LIN {X 0,Y 421.823,Z 772.372,A -85,B 0,C 180,E1 -10186.267,E2 -10186.267} C_VEL
LIN {X 0,Y 422.37,Z 759.301,A -85,B 0,C 180,E1 -10186.742,E2 -10186.742} C_VEL
LIN {X 0,Y 422.695,Z 742.091,A -85,B 0,C 180,E1 -10187.102,E2 -10187.102} C_VEL
LIN {X 0,Y 423.433,Z 672.26,A -85,B 0,C 180,E1 -10188.345,E2 -10188.345} C_VEL
LIN {X 0,Y 419.664,Z 646.445,A -85,B 0,C 180,E1 -10189.009,E2 -10189.009} C_VEL
LIN {X 0,Y 420.83,Z 628.889,A -85,B 0,C 180,E1 -10192.329,E2 -10192.329} C_VEL
LIN {X 0,Y 421.665,Z 615.532,A -85,B 0,C 180,E1 -10194.887,E2 -10194.887} C_VEL
LIN {X 0,Y 419.461,Z 603.65,A -85,B 0,C 180,E1 -10197.375,E2 -10197.375} C_VEL
LIN {X 0,Y 418.306,Z 598.381,A -85,B 0,C 180,E1 -10198.54,E2 -10198.54} C_VEL
LIN {X 0,Y 418.211,Z 598.39,A -85,B 0,C 180,E1 -10201.395,E2 -10201.395} C_VEL
LIN {X 0,Y 418.266,Z 598.386,A -85,B 0,C 180,E1 -10204.579,E2 -10204.579} C_VEL
LIN {X 0,Y 418.236,Z 598.384,A -85,B 0,C 180,E1 -10207.834,E2 -10207.834} C_VEL
LIN {X 0,Y 418.263,Z 598.383,A -85,B 0,C 180,E1 -10210.942,E2 -10210.942} C_VEL
LIN {X 0,Y 418.207,Z 598.387,A -85,B 0,C 180,E1 -10213.728,E2 -10213.728} C_VEL
LIN {X 0,Y 418.212,Z 598.391,A -85,B 0,C 180,E1 -10216.449,E2 -10216.449} C_VEL
LIN {X 0,Y 418.261,Z 598.383,A -85,B 0,C 180,E1 -10219.123,E2 -10219.123} C_VEL
LIN {X 0,Y 418.231,Z 598.385,A -85,B 0,C 180,E1 -10222.164,E2 -10222.164} C_VEL
LIN {X 0,Y 418.261,Z 598.381,A -85,B 0,C 180,E1 -10225.419,E2 -10225.419} C_VEL
LIN {X 0,Y 418.218,Z 598.389,A -85,B 0,C 180,E1 -10228.604,E2 -10228.604} C_VEL
LIN {X 0,Y 418.289,Z 598.376,A -85,B 0,C 180,E1 -10231.936,E2 -10231.936} C_VEL
LIN {X 0,Y 418.283,Z 598.383,A -85,B 0,C 180,E1 -10235.162,E2 -10235.162} C_VEL
LIN {X 0,Y 418.226,Z 598.385,A -85,B 0,C 180,E1 -10238.303,E2 -10238.303} C_VEL
LIN {X 0,Y 418.276,Z 598.382,A -85,B 0,C 180,E1 -10241.382,E2 -10241.382} C_VEL
LIN {X 0,Y 418.293,Z 598.376,A -85,B 0,C 180,E1 -10244.405,E2 -10244.405} C_VEL
LIN {X 0,Y 418.347,Z 598.375,A -85,B 0,C 180,E1 -10247.385,E2 -10247.385} C_VEL
LIN {X 0,Y 418.334,Z 598.371,A -85,B 0,C 180,E1 -10250.328,E2 -10250.328} C_VEL
LIN {X 0,Y 418.485,Z 598.359,A -85,B 0,C 180,E1 -10253.248,E2 -10253.248} C_VEL
LIN {X 0,Y 418.336,Z 598.376,A -85,B 0,C 180,E1 -10255.181,E2 -10255.181} C_VEL
LIN {X 0,Y 418.535,Z 598.347,A -85,B 0,C 180,E1 -10258.075,E2 -10258.075} C_VEL
LIN {X 0,Y 418.664,Z 598.331,A -85,B 0,C 180,E1 -10260,E2 -10260} C_VEL
LIN {X 0,Y 418.503,Z 598.351,A -85,B 0,C 180,E1 -10262.887,E2 -10262.887} C_VEL
LIN {X 0,Y 418.483,Z 598.352,A -85,B 0,C 180,E1 -10266.64,E2 -10266.64} C_VEL
LIN {X 0,Y 418.348,Z 598.377,A -85,B 0,C 180,E1 -10269.671,E2 -10269.671} C_VEL
LIN {X 0,Y 418.336,Z 598.371,A -85,B 0,C 180,E1 -10273,E2 -10273} C_VEL
LIN {X 0,Y 418.303,Z 598.375,A -85,B 0,C 180,E1 -10276.735,E2 -10276.735} C_VEL
LIN {X 0,Y 418.261,Z 598.388,A -85,B 0,C 180,E1 -10279.79,E2 -10279.79} C_VEL
LIN {X 0,Y 418.228,Z 598.384,A -85,B 0,C 180,E1 -10282.736,E2 -10282.736} C_VEL
LIN {X 0,Y 418.262,Z 598.388,A -85,B 0,C 180,E1 -10285.904,E2 -10285.904} C_VEL
LIN {X 0,Y 418.265,Z 598.38,A -85,B 0,C 180,E1 -10289.161,E2 -10289.161} C_VEL
LIN {X 0,Y 418.251,Z 598.381,A -85,B 0,C 180,E1 -10292.845,E2 -10292.845} C_VEL
LIN {X 0,Y 418.24,Z 598.389,A -85,B 0,C 180,E1 -10296.239,E2 -10296.239} C_VEL
LIN {X 0,Y 418.26,Z 598.382,A -85,B 0,C 180,E1 -10299.68,E2 -10299.68} C_VEL
LIN {X 0,Y 418.278,Z 598.384,A -85,B 0,C 180,E1 -10302.33,E2 -10302.33} C_VEL
LIN {X 0,Y 418.247,Z 598.382,A -85,B 0,C 180,E1 -10305.112,E2 -10305.112} C_VEL
LIN {X 0,Y 418.249,Z 598.383,A -85,B 0,C 180,E1 -10307.769,E2 -10307.769} C_VEL
LIN {X 0,Y 418.253,Z 598.386,A -85,B 0,C 180,E1 -10310.619,E2 -10310.619} C_VEL
LIN {X 0,Y 418.239,Z 598.385,A -85,B 0,C 180,E1 -10313.977,E2 -10313.977} C_VEL
LIN {X 0,Y 418.251,Z 598.382,A -85,B 0,C 180,E1 -10317.156,E2 -10317.156} C_VEL
LIN {X 0,Y 418.263,Z 598.383,A -85,B 0,C 180,E1 -10320.896,E2 -10320.896} C_VEL
LIN {X 0,Y 418.266,Z 598.381,A -85,B 0,C 180,E1 -10324.096,E2 -10324.096} C_VEL
LIN {X 0,Y 418.234,Z 598.385,A -85,B 0,C 180,E1 -10327.264,E2 -10327.264} C_VEL
LIN {X 0,Y 418.279,Z 598.381,A -85,B 0,C 180,E1 -10330.365,E2 -10330.365} C_VEL
LIN {X 0,Y 418.313,Z 598.375,A -85,B 0,C 180,E1 -10333.405,E2 -10333.405} C_VEL
LIN {X 0,Y 418.343,Z 598.376,A -85,B 0,C 180,E1 -10336.999,E2 -10336.999} C_VEL
LIN {X 0,Y 418.338,Z 598.372,A -85,B 0,C 180,E1 -10340.329,E2 -10340.329} C_VEL
LIN {X 0,Y 418.484,Z 598.356,A -85,B 0,C 180,E1 -10343.249,E2 -10343.249} C_VEL
LIN {X 0,Y 418.337,Z 598.376,A -85,B 0,C 180,E1 -10345.182,E2 -10345.182} C_VEL
LIN {X 0,Y 418.542,Z 598.345,A -85,B 0,C 180,E1 -10348.076,E2 -10348.076} C_VEL
LIN {X 0,Y 418.67,Z 598.329,A -85,B 0,C 180,E1 -10350,E2 -10350} C_VEL
LIN {X 0,Y 418.508,Z 598.354,A -85,B 0,C 180,E1 -10352.888,E2 -10352.888} C_VEL
LIN {X 0,Y 418.484,Z 598.355,A -85,B 0,C 180,E1 -10356.751,E2 -10356.751} C_VEL
LIN {X 0,Y 418.338,Z 598.373,A -85,B 0,C 180,E1 -10359.671,E2 -10359.671} C_VEL
LIN {X 0,Y 418.319,Z 598.376,A -85,B 0,C 180,E1 -10363.342,E2 -10363.342} C_VEL
LIN {X 0,Y 417.626,Z 598.464,A -85,B 0,C 180,E1 -10364.146,E2 -10364.146} C_VEL
LIN {X 0,Y 414.748,Z 598.824,A -85,B 0,C 180,E1 -10365.451,E2 -10365.451} C_VEL
LIN {X 0,Y 412.334,Z 599.121,A -85,B 0,C 180,E1 -10366.505,E2 -10366.505} C_VEL
LIN {X 0,Y 411.312,Z 599.253,A -85,B 0,C 180,E1 -10367.32,E2 -10367.32} C_VEL
LIN {X 0,Y 411.236,Z 599.257,A -85,B 0,C 180,E1 -10367.596,E2 -10367.596} C_VEL
LIN {X 0,Y 411.195,Z 599.266,A -85,B 0,C 180,E1 -10371.034,E2 -10371.034} C_VEL
LIN {X 0,Y 411.276,Z 599.382,A -85,B 0,C 180,E1 -10373.276,E2 -10373.276} C_VEL
LIN {X 0,Y 412.939,Z 608.733,A -85,B 0,C 180,E1 -10375.742,E2 -10375.742} C_VEL
LIN {X 0,Y 412.98,Z 609.152,A -85,B 0,C 180,E1 -10375.806,E2 -10375.806} C_VEL
LIN {X 0,Y 417.05,Z 628.232,A -85,B 0,C 180,E1 -10376.355,E2 -10376.355} C_VEL
LIN {X 0,Y 415.798,Z 716.325,A -85,B 0,C 180,E1 -10377.971,E2 -10377.971} C_VEL
LIN {X 0,Y 415.423,Z 730.048,A -85,B 0,C 180,E1 -10378.435,E2 -10378.435} C_VEL
LIN {X 0,Y 414.909,Z 742.373,A -85,B 0,C 180,E1 -10379.048,E2 -10379.048} C_VEL
LIN {X 0,Y 414.304,Z 753.409,A -85,B 0,C 180,E1 -10379.782,E2 -10379.782} C_VEL
LIN {X 0,Y 413.557,Z 765.254,A -85,B 0,C 180,E1 -10380.793,E2 -10380.793} C_VEL
LIN {X 0,Y 412.878,Z 775.146,A -85,B 0,C 180,E1 -10381.848,E2 -10381.848} C_VEL
LIN {X 0,Y 412.252,Z 784.368,A -85,B 0,C 180,E1 -10383.06,E2 -10383.06} C_VEL
LIN {X 0,Y 411.647,Z 792.069,A -85,B 0,C 180,E1 -10384.291,E2 -10384.291} C_VEL
LIN {X 0,Y 411.086,Z 799.616,A -85,B 0,C 180,E1 -10385.772,E2 -10385.772} C_VEL
LIN {X 0,Y 410.669,Z 806.242,A -85,B 0,C 180,E1 -10387.41,E2 -10387.41} C_VEL
LIN {X 0,Y 410.42,Z 810.287,A -85,B 0,C 180,E1 -10388.682,E2 -10388.682} C_VEL
LIN {X 0,Y 410.182,Z 813.761,A -85,B 0,C 180,E1 -10390.061,E2 -10390.061} C_VEL
LIN {X 0,Y 410.086,Z 815.725,A -85,B 0,C 180,E1 -10391.057,E2 -10391.057} C_VEL
LIN {X 0,Y 409.93,Z 817.771,A -85,B 0,C 180,E1 -10392.507,E2 -10392.507} C_VEL
LIN {X 0,Y 409.855,Z 818.913,A -85,B 0,C 180,E1 -10393.93,E2 -10393.93} C_VEL
LIN {X 0,Y 409.832,Z 819.229,A -85,B 0,C 180,E1 -10395.326,E2 -10395.326} C_VEL
LIN {X 0,Y 409.897,Z 818.763,A -85,B 0,C 180,E1 -10396.7,E2 -10396.7} C_VEL
LIN {X 0,Y 409.982,Z 817.509,A -85,B 0,C 180,E1 -10398.046,E2 -10398.046} C_VEL
LIN {X 0,Y 410.122,Z 815.529,A -85,B 0,C 180,E1 -10399.37,E2 -10399.37} C_VEL
LIN {X 0,Y 410.333,Z 812.826,A -85,B 0,C 180,E1 -10400.676,E2 -10400.676} C_VEL
LIN {X 0,Y 410.662,Z 808.35,A -85,B 0,C 180,E1 -10402.28,E2 -10402.28} C_VEL
LIN {X 0,Y 411.094,Z 802.074,A -85,B 0,C 180,E1 -10403.988,E2 -10403.988} C_VEL
LIN {X 0,Y 411.588,Z 795.517,A -85,B 0,C 180,E1 -10405.395,E2 -10405.395} C_VEL
LIN {X 0,Y 412.163,Z 788.243,A -85,B 0,C 180,E1 -10406.668,E2 -10406.668} C_VEL
LIN {X 0,Y 412.964,Z 778.746,A -85,B 0,C 180,E1 -10408.016,E2 -10408.016} C_VEL
LIN {X 0,Y 413.716,Z 768.239,A -85,B 0,C 180,E1 -10409.22,E2 -10409.22} C_VEL
LIN {X 0,Y 414.467,Z 757.305,A -85,B 0,C 180,E1 -10410.217,E2 -10410.217} C_VEL
LIN {X 0,Y 415.151,Z 745.506,A -85,B 0,C 180,E1 -10411.057,E2 -10411.057} C_VEL
LIN {X 0,Y 415.776,Z 732.459,A -85,B 0,C 180,E1 -10411.752,E2 -10411.752} C_VEL
LIN {X 0,Y 416.109,Z 720.19,A -85,B 0,C 180,E1 -10412.205,E2 -10412.205} C_VEL
LIN {X 0,Y 416.441,Z 702.273,A -85,B 0,C 180,E1 -10412.587,E2 -10412.587} C_VEL
LIN {X 0,Y 417.534,Z 628.412,A -85,B 0,C 180,E1 -10413.947,E2 -10413.947} C_VEL
LIN {X 0,Y 413.333,Z 610.254,A -85,B 0,C 180,E1 -10414.529,E2 -10414.529} C_VEL
LIN {X 0,Y 411.425,Z 600.35,A -85,B 0,C 180,E1 -10417.281,E2 -10417.281} C_VEL
LIN {X 0,Y 411.231,Z 599.262,A -85,B 0,C 180,E1 -10417.637,E2 -10417.637} C_VEL
LIN {X 0,Y 411.214,Z 599.263,A -85,B 0,C 180,E1 -10421.052,E2 -10421.052} C_VEL
LIN {X 0,Y 411.245,Z 599.259,A -85,B 0,C 180,E1 -10424.132,E2 -10424.132} C_VEL
LIN {X 0,Y 411.306,Z 599.251,A -85,B 0,C 180,E1 -10427.166,E2 -10427.166} C_VEL
LIN {X 0,Y 411.3,Z 599.253,A -85,B 0,C 180,E1 -10430.162,E2 -10430.162} C_VEL
LIN {X 0,Y 411.453,Z 599.234,A -85,B 0,C 180,E1 -10433.133,E2 -10433.133} C_VEL
LIN {X 0,Y 411.311,Z 599.252,A -85,B 0,C 180,E1 -10435.1,E2 -10435.1} C_VEL
LIN {X 0,Y 411.506,Z 599.224,A -85,B 0,C 180,E1 -10438.043,E2 -10438.043} C_VEL
LIN {X 0,Y 411.634,Z 599.208,A -85,B 0,C 180,E1 -10440,E2 -10440} C_VEL
LIN {X 0,Y 411.459,Z 599.233,A -85,B 0,C 180,E1 -10442.938,E2 -10442.938} C_VEL
LIN {X 0,Y 411.484,Z 599.226,A -85,B 0,C 180,E1 -10445.882,E2 -10445.882} C_VEL
LIN {X 0,Y 411.473,Z 599.228,A -85,B 0,C 180,E1 -10447.854,E2 -10447.854} C_VEL
LIN {X 0,Y 411.292,Z 599.249,A -85,B 0,C 180,E1 -10451.833,E2 -10451.833} C_VEL
LIN {X 0,Y 411.255,Z 599.259,A -85,B 0,C 180,E1 -10454.853,E2 -10454.853} C_VEL
LIN {X 0,Y 411.245,Z 599.256,A -85,B 0,C 180,E1 -10457.916,E2 -10457.916} C_VEL
LIN {X 0,Y 411.189,Z 599.268,A -85,B 0,C 180,E1 -10461.035,E2 -10461.035} C_VEL
LIN {X 0,Y 411.22,Z 599.258,A -85,B 0,C 180,E1 -10464.216,E2 -10464.216} C_VEL
LIN {X 0,Y 411.254,Z 599.256,A -85,B 0,C 180,E1 -10467.479,E2 -10467.479} C_VEL
LIN {X 0,Y 411.196,Z 599.262,A -85,B 0,C 180,E1 -10470.848,E2 -10470.848} C_VEL
LIN {X 0,Y 411.201,Z 599.258,A -85,B 0,C 180,E1 -10474.334,E2 -10474.334} C_VEL
LIN {X 0,Y 411.198,Z 599.26,A -85,B 0,C 180,E1 -10477.974,E2 -10477.974} C_VEL
LIN {X 0,Y 411.196,Z 599.263,A -85,B 0,C 180,E1 -10481.235,E2 -10481.235} C_VEL
LIN {X 0,Y 411.176,Z 599.265,A -85,B 0,C 180,E1 -10484.491,E2 -10484.491} C_VEL
LIN {X 0,Y 411.196,Z 599.264,A -85,B 0,C 180,E1 -10488.198,E2 -10488.198} C_VEL
LIN {X 0,Y 411.229,Z 599.259,A -85,B 0,C 180,E1 -10490.778,E2 -10490.778} C_VEL
LIN {X 0,Y 411.199,Z 599.263,A -85,B 0,C 180,E1 -10494.472,E2 -10494.472} C_VEL
LIN {X 0,Y 411.207,Z 599.266,A -85,B 0,C 180,E1 -10496.874,E2 -10496.874} C_VEL
LIN {X 0,Y 411.233,Z 599.26,A -85,B 0,C 180,E1 -10500.645,E2 -10500.645} C_VEL
LIN {X 0,Y 411.286,Z 599.471,A -85,B 0,C 180,E1 -10501.053,E2 -10501.053} C_VEL
LIN {X 0,Y 413.939,Z 611.637,A -85,B 0,C 180,E1 -10503.805,E2 -10503.805} C_VEL
LIN {X 0,Y 414.82,Z 618.241,A -85,B 0,C 180,E1 -10505.209,E2 -10505.209} C_VEL
LIN {X 0,Y 413.388,Z 636.622,A -85,B 0,C 180,E1 -10508.822,E2 -10508.822} C_VEL
LIN {X 0,Y 412.866,Z 645.177,A -85,B 0,C 180,E1 -10510.469,E2 -10510.469} C_VEL
LIN {X 0,Y 417.124,Z 673.617,A -85,B 0,C 180,E1 -10511.235,E2 -10511.235} C_VEL
LIN {X 0,Y 416.02,Z 754.511,A -85,B 0,C 180,E1 -10512.741,E2 -10512.741} C_VEL
LIN {X 0,Y 415.372,Z 768.188,A -85,B 0,C 180,E1 -10513.189,E2 -10513.189} C_VEL
LIN {X 0,Y 414.67,Z 781.114,A -85,B 0,C 180,E1 -10513.824,E2 -10513.824} C_VEL
LIN {X 0,Y 413.905,Z 792.923,A -85,B 0,C 180,E1 -10514.615,E2 -10514.615} C_VEL
LIN {X 0,Y 413.132,Z 804.351,A -85,B 0,C 180,E1 -10515.595,E2 -10515.595} C_VEL
LIN {X 0,Y 412.392,Z 814.69,A -85,B 0,C 180,E1 -10516.699,E2 -10516.699} C_VEL
LIN {X 0,Y 411.701,Z 823.994,A -85,B 0,C 180,E1 -10517.93,E2 -10517.93} C_VEL
LIN {X 0,Y 410.972,Z 833.067,A -85,B 0,C 180,E1 -10519.407,E2 -10519.407} C_VEL
LIN {X 0,Y 410.539,Z 840.383,A -85,B 0,C 180,E1 -10520.889,E2 -10520.889} C_VEL
LIN {X 0,Y 410.276,Z 845.327,A -85,B 0,C 180,E1 -10522.124,E2 -10522.124} C_VEL
LIN {X 0,Y 410.093,Z 850.457,A -85,B 0,C 180,E1 -10523.713,E2 -10523.713} C_VEL
LIN {X 0,Y 410.056,Z 853.819,A -85,B 0,C 180,E1 -10525.084,E2 -10525.084} C_VEL
LIN {X 0,Y 409.962,Z 855.711,A -85,B 0,C 180,E1 -10526.068,E2 -10526.068} C_VEL
LIN {X 0,Y 409.995,Z 857.137,A -85,B 0,C 180,E1 -10527.052,E2 -10527.052} C_VEL
LIN {X 0,Y 410.021,Z 858.159,A -85,B 0,C 180,E1 -10528.035,E2 -10528.035} C_VEL
LIN {X 0,Y 409.979,Z 858.782,A -85,B 0,C 180,E1 -10529.018,E2 -10529.018} C_VEL
LIN {X 0,Y 409.971,Z 858.989,A -85,B 0,C 180,E1 -10530,E2 -10530} C_VEL
LIN {X 0,Y 409.978,Z 858.761,A -85,B 0,C 180,E1 -10530.982,E2 -10530.982} C_VEL
LIN {X 0,Y 410.02,Z 858.141,A -85,B 0,C 180,E1 -10531.965,E2 -10531.965} C_VEL
LIN {X 0,Y 409.988,Z 857.119,A -85,B 0,C 180,E1 -10532.948,E2 -10532.948} C_VEL
LIN {X 0,Y 409.948,Z 855.659,A -85,B 0,C 180,E1 -10533.932,E2 -10533.932} C_VEL
LIN {X 0,Y 410.044,Z 852.644,A -85,B 0,C 180,E1 -10535.409,E2 -10535.409} C_VEL
LIN {X 0,Y 410.166,Z 848.551,A -85,B 0,C 180,E1 -10536.889,E2 -10536.889} C_VEL
LIN {X 0,Y 410.467,Z 842.25,A -85,B 0,C 180,E1 -10538.616,E2 -10538.616} C_VEL
LIN {X 0,Y 410.846,Z 835.379,A -85,B 0,C 180,E1 -10540.098,E2 -10540.098} C_VEL
LIN {X 0,Y 411.438,Z 826.818,A -85,B 0,C 180,E1 -10541.578,E2 -10541.578} C_VEL
LIN {X 0,Y 412.036,Z 818,A -85,B 0,C 180,E1 -10542.811,E2 -10542.811} C_VEL
LIN {X 0,Y 412.767,Z 807.389,A -85,B 0,C 180,E1 -10544.016,E2 -10544.016} C_VEL
LIN {X 0,Y 413.534,Z 796.314,A -85,B 0,C 180,E1 -10545.021,E2 -10545.021} C_VEL
LIN {X 0,Y 414.342,Z 784.169,A -85,B 0,C 180,E1 -10545.873,E2 -10545.873} C_VEL
LIN {X 0,Y 414.923,Z 772.813,A -85,B 0,C 180,E1 -10546.481,E2 -10546.481} C_VEL
LIN {X 0,Y 415.475,Z 760.218,A -85,B 0,C 180,E1 -10546.965,E2 -10546.965} C_VEL
LIN {X 0,Y 415.812,Z 745.574,A -85,B 0,C 180,E1 -10547.299,E2 -10547.299} C_VEL
LIN {X 0,Y 416.667,Z 673.287,A -85,B 0,C 180,E1 -10548.607,E2 -10548.607} C_VEL
LIN {X 0,Y 412.721,Z 646.227,A -85,B 0,C 180,E1 -10549.305,E2 -10549.305} C_VEL
LIN {X 0,Y 413.879,Z 629.809,A -85,B 0,C 180,E1 -10552.461,E2 -10552.461} C_VEL
LIN {X 0,Y 414.722,Z 617.813,A -85,B 0,C 180,E1 -10554.797,E2 -10554.797} C_VEL
LIN {X 0,Y 413.731,Z 611.057,A -85,B 0,C 180,E1 -10556.209,E2 -10556.209} C_VEL
LIN {X 0,Y 411.259,Z 599.258,A -85,B 0,C 180,E1 -10558.798,E2 -10558.798} C_VEL
LIN {X 0,Y 411.165,Z 599.271,A -85,B 0,C 180,E1 -10561.996,E2 -10561.996} C_VEL
LIN {X 0,Y 411.211,Z 599.261,A -85,B 0,C 180,E1 -10564.878,E2 -10564.878} C_VEL
LIN {X 0,Y 411.213,Z 599.261,A -85,B 0,C 180,E1 -10568.169,E2 -10568.169} C_VEL
LIN {X 0,Y 411.198,Z 599.261,A -85,B 0,C 180,E1 -10571.233,E2 -10571.233} C_VEL
LIN {X 0,Y 411.174,Z 599.269,A -85,B 0,C 180,E1 -10574.489,E2 -10574.489} C_VEL
LIN {X 0,Y 411.196,Z 599.262,A -85,B 0,C 180,E1 -10578.196,E2 -10578.196} C_VEL
LIN {X 0,Y 411.224,Z 599.264,A -85,B 0,C 180,E1 -10580.776,E2 -10580.776} C_VEL
LIN {X 0,Y 411.195,Z 599.264,A -85,B 0,C 180,E1 -10584.47,E2 -10584.47} C_VEL
LIN {X 0,Y 411.167,Z 599.264,A -85,B 0,C 180,E1 -10588.002,E2 -10588.002} C_VEL
LIN {X 0,Y 411.218,Z 599.26,A -85,B 0,C 180,E1 -10591.409,E2 -10591.409} C_VEL
LIN {X 0,Y 411.23,Z 599.26,A -85,B 0,C 180,E1 -10594.706,E2 -10594.706} C_VEL
LIN {X 0,Y 411.197,Z 599.26,A -85,B 0,C 180,E1 -10597.912,E2 -10597.912} C_VEL
LIN {X 0,Y 411.217,Z 599.264,A -85,B 0,C 180,E1 -10601.051,E2 -10601.051} C_VEL
LIN {X 0,Y 411.246,Z 599.254,A -85,B 0,C 180,E1 -10604.131,E2 -10604.131} C_VEL
LIN {X 0,Y 411.295,Z 599.255,A -85,B 0,C 180,E1 -10607.165,E2 -10607.165} C_VEL
LIN {X 0,Y 411.286,Z 599.249,A -85,B 0,C 180,E1 -10610.161,E2 -10610.161} C_VEL
LIN {X 0,Y 411.448,Z 599.234,A -85,B 0,C 180,E1 -10613.132,E2 -10613.132} C_VEL
LIN {X 0,Y 411.306,Z 599.251,A -85,B 0,C 180,E1 -10615.098,E2 -10615.098} C_VEL
LIN {X 0,Y 411.505,Z 599.223,A -85,B 0,C 180,E1 -10618.042,E2 -10618.042} C_VEL
LIN {X 0,Y 411.634,Z 599.207,A -85,B 0,C 180,E1 -10620,E2 -10620} C_VEL
LIN {X 0,Y 411.459,Z 599.229,A -85,B 0,C 180,E1 -10622.937,E2 -10622.937} C_VEL
LIN {X 0,Y 411.445,Z 599.229,A -85,B 0,C 180,E1 -10626.639,E2 -10626.639} C_VEL
LIN {X 0,Y 411.295,Z 599.253,A -85,B 0,C 180,E1 -10629.838,E2 -10629.838} C_VEL
LIN {X 0,Y 411.295,Z 599.249,A -85,B 0,C 180,E1 -10633.104,E2 -10633.104} C_VEL
LIN {X 0,Y 411.247,Z 599.254,A -85,B 0,C 180,E1 -10636.889,E2 -10636.889} C_VEL
LIN {X 0,Y 411.221,Z 599.263,A -85,B 0,C 180,E1 -10639.987,E2 -10639.987} C_VEL
LIN {X 0,Y 411.193,Z 599.261,A -85,B 0,C 180,E1 -10643.148,E2 -10643.148} C_VEL
LIN {X 0,Y 411.229,Z 599.258,A -85,B 0,C 180,E1 -10646.381,E2 -10646.381} C_VEL
LIN {X 0,Y 411.202,Z 599.263,A -85,B 0,C 180,E1 -10649.712,E2 -10649.712} C_VEL
LIN {X 0,Y 411.198,Z 599.26,A -85,B 0,C 180,E1 -10653.156,E2 -10653.156} C_VEL
LIN {X 0,Y 411.187,Z 599.264,A -85,B 0,C 180,E1 -10656.553,E2 -10656.553} C_VEL
LIN {X 0,Y 411.222,Z 599.259,A -85,B 0,C 180,E1 -10659.731,E2 -10659.731} C_VEL
LIN {X 0,Y 411.217,Z 599.257,A -85,B 0,C 180,E1 -10663.127,E2 -10663.127} C_VEL
LIN {X 0,Y 411.169,Z 599.266,A -85,B 0,C 180,E1 -10665.88,E2 -10665.88} C_VEL
LIN {X 0,Y 411.19,Z 599.263,A -85,B 0,C 180,E1 -10668.767,E2 -10668.767} C_VEL
LIN {X 0,Y 411.194,Z 599.263,A -85,B 0,C 180,E1 -10672.027,E2 -10672.027} C_VEL
LIN {X 0,Y 411.2,Z 599.26,A -85,B 0,C 180,E1 -10675.667,E2 -10675.667} C_VEL
LIN {X 0,Y 411.183,Z 599.263,A -85,B 0,C 180,E1 -10679.153,E2 -10679.153} C_VEL
LIN {X 0,Y 411.254,Z 599.26,A -85,B 0,C 180,E1 -10682.523,E2 -10682.523} C_VEL
LIN {X 0,Y 411.222,Z 599.257,A -85,B 0,C 180,E1 -10685.785,E2 -10685.785} C_VEL
LIN {X 0,Y 411.192,Z 599.265,A -85,B 0,C 180,E1 -10688.966,E2 -10688.966} C_VEL
LIN {X 0,Y 411.249,Z 599.254,A -85,B 0,C 180,E1 -10692.085,E2 -10692.085} C_VEL
LIN {X 0,Y 411.259,Z 599.256,A -85,B 0,C 180,E1 -10695.148,E2 -10695.148} C_VEL
LIN {X 0,Y 411.281,Z 599.25,A -85,B 0,C 180,E1 -10698.167,E2 -10698.167} C_VEL
LIN {X 0,Y 411.437,Z 599.231,A -85,B 0,C 180,E1 -10702.189,E2 -10702.189} C_VEL
LIN {X 0,Y 411.468,Z 599.226,A -85,B 0,C 180,E1 -10704.118,E2 -10704.118} C_VEL
LIN {X 0,Y 411.511,Z 599.221,A -85,B 0,C 180,E1 -10708.043,E2 -10708.043} C_VEL
LIN {X 0,Y 411.639,Z 599.205,A -85,B 0,C 180,E1 -10710,E2 -10710} C_VEL
LIN {X 0,Y 411.464,Z 599.232,A -85,B 0,C 180,E1 -10712.937,E2 -10712.937} C_VEL
LIN {X 0,Y 411.448,Z 599.232,A -85,B 0,C 180,E1 -10716.867,E2 -10716.867} C_VEL
LIN {X 0,Y 411.29,Z 599.25,A -85,B 0,C 180,E1 -10719.839,E2 -10719.839} C_VEL
LIN {X 0,Y 411.279,Z 599.253,A -85,B 0,C 180,E1 -10723.33,E2 -10723.33} C_VEL
LIN {X 0,Y 411.253,Z 599.255,A -85,B 0,C 180,E1 -10726.888,E2 -10726.888} C_VEL
LIN {X 0,Y 411.236,Z 599.257,A -85,B 0,C 180,E1 -10727.596,E2 -10727.596} C_VEL
LIN {X 0,Y 410.58,Z 599.343,A -85,B 0,C 180,E1 -10728.414,E2 -10728.414} C_VEL
LIN {X 0,Y 407.705,Z 599.704,A -85,B 0,C 180,E1 -10729.742,E2 -10729.742} C_VEL
LIN {X 0,Y 405.269,Z 600.006,A -85,B 0,C 180,E1 -10730.815,E2 -10730.815} C_VEL
LIN {X 0,Y 404.233,Z 600.133,A -85,B 0,C 180,E1 -10731.645,E2 -10731.645} C_VEL
LIN {X 0,Y 404.154,Z 600.141,A -85,B 0,C 180,E1 -10731.926,E2 -10731.926} C_VEL
LIN {X 0,Y 404.188,Z 600.162,A -85,B 0,C 180,E1 -10733.034,E2 -10733.034} C_VEL
LIN {X 0,Y 405.884,Z 609.284,A -85,B 0,C 180,E1 -10735.478,E2 -10735.478} C_VEL
LIN {X 0,Y 410.345,Z 629.499,A -85,B 0,C 180,E1 -10736.076,E2 -10736.076} C_VEL
LIN {X 0,Y 408.991,Z 716.33,A -85,B 0,C 180,E1 -10737.694,E2 -10737.694} C_VEL
LIN {X 0,Y 408.575,Z 730.058,A -85,B 0,C 180,E1 -10738.161,E2 -10738.161} C_VEL
LIN {X 0,Y 408.106,Z 741.751,A -85,B 0,C 180,E1 -10738.744,E2 -10738.744} C_VEL
LIN {X 0,Y 407.502,Z 752.388,A -85,B 0,C 180,E1 -10739.44,E2 -10739.44} C_VEL
LIN {X 0,Y 406.765,Z 764.197,A -85,B 0,C 180,E1 -10740.438,E2 -10740.438} C_VEL
LIN {X 0,Y 405.951,Z 775.434,A -85,B 0,C 180,E1 -10741.639,E2 -10741.639} C_VEL
LIN {X 0,Y 405.245,Z 785.274,A -85,B 0,C 180,E1 -10742.964,E2 -10742.964} C_VEL
LIN {X 0,Y 404.542,Z 793.751,A -85,B 0,C 180,E1 -10744.374,E2 -10744.374} C_VEL
LIN {X 0,Y 403.951,Z 801.521,A -85,B 0,C 180,E1 -10745.985,E2 -10745.985} C_VEL
LIN {X 0,Y 403.583,Z 807.429,A -85,B 0,C 180,E1 -10747.552,E2 -10747.552} C_VEL
LIN {X 0,Y 403.215,Z 812.694,A -85,B 0,C 180,E1 -10749.379,E2 -10749.379} C_VEL
LIN {X 0,Y 403.031,Z 815.673,A -85,B 0,C 180,E1 -10750.791,E2 -10750.791} C_VEL
LIN {X 0,Y 402.955,Z 816.856,A -85,B 0,C 180,E1 -10751.51,E2 -10751.51} C_VEL
LIN {X 0,Y 402.828,Z 818.524,A -85,B 0,C 180,E1 -10752.883,E2 -10752.883} C_VEL
LIN {X 0,Y 402.769,Z 819.451,A -85,B 0,C 180,E1 -10754.323,E2 -10754.323} C_VEL
LIN {X 0,Y 402.774,Z 819.522,A -85,B 0,C 180,E1 -10755.737,E2 -10755.737} C_VEL
LIN {X 0,Y 402.83,Z 818.82,A -85,B 0,C 180,E1 -10757.125,E2 -10757.125} C_VEL
LIN {X 0,Y 402.968,Z 817.251,A -85,B 0,C 180,E1 -10758.584,E2 -10758.584} C_VEL
LIN {X 0,Y 403.142,Z 814.702,A -85,B 0,C 180,E1 -10760.088,E2 -10760.088} C_VEL
LIN {X 0,Y 403.435,Z 811.066,A -85,B 0,C 180,E1 -10761.619,E2 -10761.619} C_VEL
LIN {X 0,Y 403.854,Z 805.176,A -85,B 0,C 180,E1 -10763.459,E2 -10763.459} C_VEL
LIN {X 0,Y 404.387,Z 798.74,A -85,B 0,C 180,E1 -10765.005,E2 -10765.005} C_VEL
LIN {X 0,Y 404.962,Z 791.446,A -85,B 0,C 180,E1 -10766.409,E2 -10766.409} C_VEL
LIN {X 0,Y 405.817,Z 782.357,A -85,B 0,C 180,E1 -10767.819,E2 -10767.819} C_VEL
LIN {X 0,Y 406.549,Z 772.938,A -85,B 0,C 180,E1 -10769.01,E2 -10769.01} C_VEL
LIN {X 0,Y 407.374,Z 761.947,A -85,B 0,C 180,E1 -10770.123,E2 -10770.123} C_VEL
LIN {X 0,Y 408.171,Z 749.52,A -85,B 0,C 180,E1 -10771.107,E2 -10771.107} C_VEL
LIN {X 0,Y 408.827,Z 738.228,A -85,B 0,C 180,E1 -10771.788,E2 -10771.788} C_VEL
LIN {X 0,Y 409.175,Z 724.979,A -85,B 0,C 180,E1 -10772.371,E2 -10772.371} C_VEL
LIN {X 0,Y 409.597,Z 712.282,A -85,B 0,C 180,E1 -10772.718,E2 -10772.718} C_VEL
LIN {X 0,Y 410.918,Z 629.538,A -85,B 0,C 180,E1 -10774.274,E2 -10774.274} C_VEL
LIN {X 0,Y 406.957,Z 612.65,A -85,B 0,C 180,E1 -10774.833,E2 -10774.833} C_VEL
LIN {X 0,Y 406.309,Z 610.6,A -85,B 0,C 180,E1 -10774.927,E2 -10774.927} C_VEL
LIN {X 0,Y 404.195,Z 600.14,A -85,B 0,C 180,E1 -10777.914,E2 -10777.914} C_VEL
LIN {X 0,Y 404.156,Z 600.144,A -85,B 0,C 180,E1 -10780.708,E2 -10780.708} C_VEL
LIN {X 0,Y 404.212,Z 600.134,A -85,B 0,C 180,E1 -10783.848,E2 -10783.848} C_VEL
LIN {X 0,Y 404.273,Z 600.128,A -85,B 0,C 180,E1 -10786.939,E2 -10786.939} C_VEL
LIN {X 0,Y 404.263,Z 600.128,A -85,B 0,C 180,E1 -10789.989,E2 -10789.989} C_VEL
LIN {X 0,Y 404.404,Z 600.114,A -85,B 0,C 180,E1 -10793.013,E2 -10793.013} C_VEL
LIN {X 0,Y 404.283,Z 600.129,A -85,B 0,C 180,E1 -10795.014,E2 -10795.014} C_VEL
LIN {X 0,Y 404.475,Z 600.1,A -85,B 0,C 180,E1 -10798.009,E2 -10798.009} C_VEL
LIN {X 0,Y 404.604,Z 600.084,A -85,B 0,C 180,E1 -10800.001,E2 -10800.001} C_VEL
LIN {X 0,Y 404.417,Z 600.11,A -85,B 0,C 180,E1 -10802.989,E2 -10802.989} C_VEL
LIN {X 0,Y 404.43,Z 600.104,A -85,B 0,C 180,E1 -10805.985,E2 -10805.985} C_VEL
LIN {X 0,Y 404.415,Z 600.107,A -85,B 0,C 180,E1 -10807.992,E2 -10807.992} C_VEL
LIN {X 0,Y 404.263,Z 600.125,A -85,B 0,C 180,E1 -10812.042,E2 -10812.042} C_VEL
LIN {X 0,Y 404.2,Z 600.135,A -85,B 0,C 180,E1 -10815.119,E2 -10815.119} C_VEL
LIN {X 0,Y 404.202,Z 600.133,A -85,B 0,C 180,E1 -10818.239,E2 -10818.239} C_VEL
LIN {X 0,Y 404.131,Z 600.143,A -85,B 0,C 180,E1 -10821.42,E2 -10821.42} C_VEL
LIN {X 0,Y 404.171,Z 600.138,A -85,B 0,C 180,E1 -10824.667,E2 -10824.667} C_VEL
LIN {X 0,Y 404.192,Z 600.132,A -85,B 0,C 180,E1 -10828,E2 -10828} C_VEL
LIN {X 0,Y 404.142,Z 600.138,A -85,B 0,C 180,E1 -10831.561,E2 -10831.561} C_VEL
LIN {X 0,Y 404.181,Z 600.135,A -85,B 0,C 180,E1 -10835.017,E2 -10835.017} C_VEL
LIN {X 0,Y 404.157,Z 600.137,A -85,B 0,C 180,E1 -10838.757,E2 -10838.757} C_VEL
LIN {X 0,Y 404.147,Z 600.144,A -85,B 0,C 180,E1 -10841.605,E2 -10841.605} C_VEL
LIN {X 0,Y 404.146,Z 600.141,A -85,B 0,C 180,E1 -10844.524,E2 -10844.524} C_VEL
LIN {X 0,Y 404.168,Z 600.143,A -85,B 0,C 180,E1 -10847.301,E2 -10847.301} C_VEL
LIN {X 0,Y 404.167,Z 600.14,A -85,B 0,C 180,E1 -10849.956,E2 -10849.956} C_VEL
LIN {X 0,Y 404.14,Z 600.145,A -85,B 0,C 180,E1 -10853.125,E2 -10853.125} C_VEL
LIN {X 0,Y 404.145,Z 600.147,A -85,B 0,C 180,E1 -10856.189,E2 -10856.189} C_VEL
LIN {X 0,Y 404.146,Z 600.145,A -85,B 0,C 180,E1 -10859.716,E2 -10859.716} C_VEL
LIN {X 0,Y 404.233,Z 600.334,A -85,B 0,C 180,E1 -10860.699,E2 -10860.699} C_VEL
LIN {X 0,Y 407.05,Z 613.117,A -85,B 0,C 180,E1 -10863.663,E2 -10863.663} C_VEL
LIN {X 0,Y 407.914,Z 619.37,A -85,B 0,C 180,E1 -10865.033,E2 -10865.033} C_VEL
LIN {X 0,Y 406.431,Z 637.74,A -85,B 0,C 180,E1 -10868.708,E2 -10868.708} C_VEL
LIN {X 0,Y 405.988,Z 644.664,A -85,B 0,C 180,E1 -10870.077,E2 -10870.077} C_VEL
LIN {X 0,Y 410.108,Z 671.961,A -85,B 0,C 180,E1 -10870.853,E2 -10870.853} C_VEL
LIN {X 0,Y 410.426,Z 676.297,A -85,B 0,C 180,E1 -10870.954,E2 -10870.954} C_VEL
LIN {X 0,Y 409.247,Z 754.77,A -85,B 0,C 180,E1 -10872.447,E2 -10872.447} C_VEL
LIN {X 0,Y 408.591,Z 768.231,A -85,B 0,C 180,E1 -10872.902,E2 -10872.902} C_VEL
LIN {X 0,Y 407.856,Z 781.013,A -85,B 0,C 180,E1 -10873.547,E2 -10873.547} C_VEL
LIN {X 0,Y 407.051,Z 792.767,A -85,B 0,C 180,E1 -10874.349,E2 -10874.349} C_VEL
LIN {X 0,Y 406.237,Z 804.157,A -85,B 0,C 180,E1 -10875.345,E2 -10875.345} C_VEL
LIN {X 0,Y 405.441,Z 814.746,A -85,B 0,C 180,E1 -10876.506,E2 -10876.506} C_VEL
LIN {X 0,Y 404.736,Z 823.719,A -85,B 0,C 180,E1 -10877.719,E2 -10877.719} C_VEL
LIN {X 0,Y 403.955,Z 832.769,A -85,B 0,C 180,E1 -10879.221,E2 -10879.221} C_VEL
LIN {X 0,Y 403.49,Z 840.072,A -85,B 0,C 180,E1 -10880.729,E2 -10880.729} C_VEL
LIN {X 0,Y 403.212,Z 845.013,A -85,B 0,C 180,E1 -10881.985,E2 -10881.985} C_VEL
LIN {X 0,Y 402.987,Z 850.553,A -85,B 0,C 180,E1 -10883.759,E2 -10883.759} C_VEL
LIN {X 0,Y 402.964,Z 853.496,A -85,B 0,C 180,E1 -10884.997,E2 -10884.997} C_VEL
LIN {X 0,Y 402.882,Z 855.382,A -85,B 0,C 180,E1 -10885.999,E2 -10885.999} C_VEL
LIN {X 0,Y 402.894,Z 856.803,A -85,B 0,C 180,E1 -10887,E2 -10887} C_VEL
LIN {X 0,Y 402.95,Z 857.824,A -85,B 0,C 180,E1 -10888.001,E2 -10888.001} C_VEL
LIN {X 0,Y 402.904,Z 858.444,A -85,B 0,C 180,E1 -10889.001,E2 -10889.001} C_VEL
LIN {X 0,Y 402.894,Z 858.641,A -85,B 0,C 180,E1 -10890,E2 -10890} C_VEL
LIN {X 0,Y 402.904,Z 858.408,A -85,B 0,C 180,E1 -10890.999,E2 -10890.999} C_VEL
LIN {X 0,Y 402.949,Z 857.783,A -85,B 0,C 180,E1 -10891.999,E2 -10891.999} C_VEL
LIN {X 0,Y 402.888,Z 856.753,A -85,B 0,C 180,E1 -10893,E2 -10893} C_VEL
LIN {X 0,Y 402.869,Z 855.281,A -85,B 0,C 180,E1 -10894.001,E2 -10894.001} C_VEL
LIN {X 0,Y 402.943,Z 852.249,A -85,B 0,C 180,E1 -10895.505,E2 -10895.505} C_VEL
LIN {X 0,Y 403.078,Z 848.139,A -85,B 0,C 180,E1 -10897.01,E2 -10897.01} C_VEL
LIN {X 0,Y 403.402,Z 841.816,A -85,B 0,C 180,E1 -10898.768,E2 -10898.768} C_VEL
LIN {X 0,Y 403.792,Z 834.921,A -85,B 0,C 180,E1 -10900.276,E2 -10900.276} C_VEL
LIN {X 0,Y 404.426,Z 826.32,A -85,B 0,C 180,E1 -10901.782,E2 -10901.782} C_VEL
LIN {X 0,Y 405.064,Z 817.468,A -85,B 0,C 180,E1 -10903.035,E2 -10903.035} C_VEL
LIN {X 0,Y 405.837,Z 806.575,A -85,B 0,C 180,E1 -10904.286,E2 -10904.286} C_VEL
LIN {X 0,Y 406.63,Z 795.657,A -85,B 0,C 180,E1 -10905.282,E2 -10905.282} C_VEL
LIN {X 0,Y 407.497,Z 783.435,A -85,B 0,C 180,E1 -10906.147,E2 -10906.147} C_VEL
LIN {X 0,Y 408.099,Z 771.96,A -85,B 0,C 180,E1 -10906.765,E2 -10906.765} C_VEL
LIN {X 0,Y 408.684,Z 759.087,A -85,B 0,C 180,E1 -10907.256,E2 -10907.256} C_VEL
LIN {X 0,Y 409.013,Z 743.885,A -85,B 0,C 180,E1 -10907.596,E2 -10907.596} C_VEL
LIN {X 0,Y 409.836,Z 673.84,A -85,B 0,C 180,E1 -10908.891,E2 -10908.891} C_VEL
LIN {X 0,Y 405.802,Z 645.842,A -85,B 0,C 180,E1 -10909.637,E2 -10909.637} C_VEL
LIN {X 0,Y 406.989,Z 629.393,A -85,B 0,C 180,E1 -10912.863,E2 -10912.863} C_VEL
LIN {X 0,Y 407.793,Z 618.727,A -85,B 0,C 180,E1 -10914.975,E2 -10914.975} C_VEL
LIN {X 0,Y 405.921,Z 607.889,A -85,B 0,C 180,E1 -10917.31,E2 -10917.31} C_VEL
LIN {X 0,Y 404.217,Z 600.136,A -85,B 0,C 180,E1 -10919.06,E2 -10919.06} C_VEL
LIN {X 0,Y 404.141,Z 600.146,A -85,B 0,C 180,E1 -10922.621,E2 -10922.621} C_VEL
LIN {X 0,Y 404.181,Z 600.134,A -85,B 0,C 180,E1 -10925.189,E2 -10925.189} C_VEL
LIN {X 0,Y 404.161,Z 600.141,A -85,B 0,C 180,E1 -10928.755,E2 -10928.755} C_VEL
LIN {X 0,Y 404.148,Z 600.138,A -85,B 0,C 180,E1 -10931.603,E2 -10931.603} C_VEL
LIN {X 0,Y 404.143,Z 600.145,A -85,B 0,C 180,E1 -10934.521,E2 -10934.521} C_VEL
LIN {X 0,Y 404.17,Z 600.136,A -85,B 0,C 180,E1 -10937.299,E2 -10937.299} C_VEL
LIN {X 0,Y 404.165,Z 600.136,A -85,B 0,C 180,E1 -10939.954,E2 -10939.954} C_VEL
LIN {X 0,Y 404.136,Z 600.143,A -85,B 0,C 180,E1 -10943.123,E2 -10943.123} C_VEL
LIN {X 0,Y 404.14,Z 600.14,A -85,B 0,C 180,E1 -10946.187,E2 -10946.187} C_VEL
LIN {X 0,Y 404.151,Z 600.138,A -85,B 0,C 180,E1 -10949.715,E2 -10949.715} C_VEL
LIN {X 0,Y 404.19,Z 600.139,A -85,B 0,C 180,E1 -10953.122,E2 -10953.122} C_VEL
LIN {X 0,Y 404.167,Z 600.139,A -85,B 0,C 180,E1 -10955.333,E2 -10955.333} C_VEL
LIN {X 0,Y 404.131,Z 600.142,A -85,B 0,C 180,E1 -10958.58,E2 -10958.58} C_VEL
LIN {X 0,Y 404.203,Z 600.132,A -85,B 0,C 180,E1 -10961.761,E2 -10961.761} C_VEL
LIN {X 0,Y 404.197,Z 600.136,A -85,B 0,C 180,E1 -10964.881,E2 -10964.881} C_VEL
LIN {X 0,Y 404.249,Z 600.126,A -85,B 0,C 180,E1 -10967.958,E2 -10967.958} C_VEL
LIN {X 0,Y 404.397,Z 600.107,A -85,B 0,C 180,E1 -10972.128,E2 -10972.128} C_VEL
LIN {X 0,Y 404.416,Z 600.105,A -85,B 0,C 180,E1 -10974.014,E2 -10974.014} C_VEL
LIN {X 0,Y 404.474,Z 600.099,A -85,B 0,C 180,E1 -10978.008,E2 -10978.008} C_VEL
LIN {X 0,Y 404.604,Z 600.083,A -85,B 0,C 180,E1 -10979.999,E2 -10979.999} C_VEL
LIN {X 0,Y 404.416,Z 600.107,A -85,B 0,C 180,E1 -10982.988,E2 -10982.988} C_VEL
LIN {X 0,Y 404.392,Z 600.108,A -85,B 0,C 180,E1 -10986.637,E2 -10986.637} C_VEL
LIN {X 0,Y 404.285,Z 600.122,A -85,B 0,C 180,E1 -10989.001,E2 -10989.001} C_VEL
LIN {X 0,Y 404.247,Z 600.129,A -85,B 0,C 180,E1 -10992.041,E2 -10992.041} C_VEL
LIN {X 0,Y 404.196,Z 600.133,A -85,B 0,C 180,E1 -10995.118,E2 -10995.118} C_VEL
LIN {X 0,Y 404.2,Z 600.134,A -85,B 0,C 180,E1 -10998.238,E2 -10998.238} C_VEL
LIN {X 0,Y 404.129,Z 600.143,A -85,B 0,C 180,E1 -11001.419,E2 -11001.419} C_VEL
LIN {X 0,Y 404.167,Z 600.136,A -85,B 0,C 180,E1 -11004.666,E2 -11004.666} C_VEL
LIN {X 0,Y 404.189,Z 600.14,A -85,B 0,C 180,E1 -11008,E2 -11008} C_VEL
LIN {X 0,Y 404.137,Z 600.142,A -85,B 0,C 180,E1 -11011.56,E2 -11011.56} C_VEL
LIN {X 0,Y 404.177,Z 600.135,A -85,B 0,C 180,E1 -11015.016,E2 -11015.016} C_VEL
LIN {X 0,Y 404.156,Z 600.138,A -85,B 0,C 180,E1 -11018.756,E2 -11018.756} C_VEL
LIN {X 0,Y 404.184,Z 600.135,A -85,B 0,C 180,E1 -11021.611,E2 -11021.611} C_VEL
LIN {X 0,Y 404.185,Z 600.138,A -85,B 0,C 180,E1 -11024.529,E2 -11024.529} C_VEL
LIN {X 0,Y 404.165,Z 600.136,A -85,B 0,C 180,E1 -11027.301,E2 -11027.301} C_VEL
LIN {X 0,Y 404.162,Z 600.139,A -85,B 0,C 180,E1 -11029.956,E2 -11029.956} C_VEL
LIN {X 0,Y 404.133,Z 600.141,A -85,B 0,C 180,E1 -11033.125,E2 -11033.125} C_VEL
LIN {X 0,Y 404.139,Z 600.143,A -85,B 0,C 180,E1 -11036.188,E2 -11036.188} C_VEL
LIN {X 0,Y 404.14,Z 600.139,A -85,B 0,C 180,E1 -11039.715,E2 -11039.715} C_VEL
LIN {X 0,Y 404.19,Z 600.135,A -85,B 0,C 180,E1 -11043.123,E2 -11043.123} C_VEL
LIN {X 0,Y 404.172,Z 600.136,A -85,B 0,C 180,E1 -11045.335,E2 -11045.335} C_VEL
LIN {X 0,Y 404.155,Z 600.143,A -85,B 0,C 180,E1 -11048.582,E2 -11048.582} C_VEL
LIN {X 0,Y 404.206,Z 600.131,A -85,B 0,C 180,E1 -11051.762,E2 -11051.762} C_VEL
LIN {X 0,Y 404.205,Z 600.138,A -85,B 0,C 180,E1 -11054.882,E2 -11054.882} C_VEL
LIN {X 0,Y 404.253,Z 600.125,A -85,B 0,C 180,E1 -11057.959,E2 -11057.959} C_VEL
LIN {X 0,Y 404.401,Z 600.107,A -85,B 0,C 180,E1 -11062.129,E2 -11062.129} C_VEL
LIN {X 0,Y 404.416,Z 600.105,A -85,B 0,C 180,E1 -11064.015,E2 -11064.015} C_VEL
LIN {X 0,Y 404.48,Z 600.097,A -85,B 0,C 180,E1 -11068.009,E2 -11068.009} C_VEL
LIN {X 0,Y 404.609,Z 600.081,A -85,B 0,C 180,E1 -11070,E2 -11070} C_VEL
LIN {X 0,Y 404.421,Z 600.11,A -85,B 0,C 180,E1 -11072.988,E2 -11072.988} C_VEL
LIN {X 0,Y 404.396,Z 600.112,A -85,B 0,C 180,E1 -11076.987,E2 -11076.987} C_VEL
LIN {X 0,Y 404.255,Z 600.125,A -85,B 0,C 180,E1 -11080.012,E2 -11080.012} C_VEL
LIN {X 0,Y 404.263,Z 600.13,A -85,B 0,C 180,E1 -11083.211,E2 -11083.211} C_VEL
LIN {X 0,Y 404.212,Z 600.133,A -85,B 0,C 180,E1 -11087.007,E2 -11087.007} C_VEL
LIN {X 0,Y 404.16,Z 600.141,A -85,B 0,C 180,E1 -11090.351,E2 -11090.351} C_VEL
LIN {X 0,Y 404.154,Z 600.141,A -85,B 0,C 180,E1 -11091.926,E2 -11091.926} C_VEL
LIN {X 0,Y 403.556,Z 600.581,A -85,B 0,C 180,E1 -11092.479,E2 -11092.479} C_VEL
LIN {X 0,Y 401.638,Z 602.169,A -85,B 0,C 180,E1 -11093.16,E2 -11093.16} C_VEL
LIN {X 0,Y 398.775,Z 605.761,A -85,B 0,C 180,E1 -11094.137,E2 -11094.137} C_VEL
LIN {X 0,Y 398.449,Z 607.727,A -85,B 0,C 180,E1 -11094.647,E2 -11094.647} C_VEL
LIN {X 0,Y 398.773,Z 609.501,A -85,B 0,C 180,E1 -11095.127,E2 -11095.127} C_VEL
LIN {X 0,Y 401.404,Z 619.751,A -85,B 0,C 180,E1 -11095.47,E2 -11095.47} C_VEL
LIN {X 0,Y 403.616,Z 631.346,A -85,B 0,C 180,E1 -11095.805,E2 -11095.805} C_VEL
LIN {X 0,Y 402.176,Z 716.682,A -85,B 0,C 180,E1 -11097.424,E2 -11097.424} C_VEL
LIN {X 0,Y 401.734,Z 730.273,A -85,B 0,C 180,E1 -11097.893,E2 -11097.893} C_VEL
LIN {X 0,Y 401.215,Z 742.882,A -85,B 0,C 180,E1 -11098.537,E2 -11098.537} C_VEL
LIN {X 0,Y 400.545,Z 754.396,A -85,B 0,C 180,E1 -11099.331,E2 -11099.331} C_VEL
LIN {X 0,Y 399.708,Z 766.52,A -85,B 0,C 180,E1 -11100.407,E2 -11100.407} C_VEL
LIN {X 0,Y 398.89,Z 777.196,A -85,B 0,C 180,E1 -11101.611,E2 -11101.611} C_VEL
LIN {X 0,Y 398.208,Z 786.456,A -85,B 0,C 180,E1 -11102.911,E2 -11102.911} C_VEL
LIN {X 0,Y 397.452,Z 795.403,A -85,B 0,C 180,E1 -11104.46,E2 -11104.46} C_VEL
LIN {X 0,Y 396.876,Z 802.736,A -85,B 0,C 180,E1 -11106.071,E2 -11106.071} C_VEL
LIN {X 0,Y 396.467,Z 808.592,A -85,B 0,C 180,E1 -11107.701,E2 -11107.701} C_VEL
LIN {X 0,Y 396.172,Z 812.692,A -85,B 0,C 180,E1 -11109.163,E2 -11109.163} C_VEL
LIN {X 0,Y 395.912,Z 816.581,A -85,B 0,C 180,E1 -11111.055,E2 -11111.055} C_VEL
LIN {X 0,Y 395.762,Z 818.435,A -85,B 0,C 180,E1 -11112.438,E2 -11112.438} C_VEL
LIN {X 0,Y 395.692,Z 819.559,A -85,B 0,C 180,E1 -11113.842,E2 -11113.842} C_VEL
LIN {X 0,Y 395.661,Z 819.936,A -85,B 0,C 180,E1 -11115.275,E2 -11115.275} C_VEL
LIN {X 0,Y 395.715,Z 819.499,A -85,B 0,C 180,E1 -11116.732,E2 -11116.732} C_VEL
LIN {X 0,Y 395.836,Z 818.18,A -85,B 0,C 180,E1 -11118.218,E2 -11118.218} C_VEL
LIN {X 0,Y 396.007,Z 815.926,A -85,B 0,C 180,E1 -11119.739,E2 -11119.739} C_VEL
LIN {X 0,Y 396.302,Z 812.637,A -85,B 0,C 180,E1 -11121.286,E2 -11121.286} C_VEL
LIN {X 0,Y 396.664,Z 807.859,A -85,B 0,C 180,E1 -11122.958,E2 -11122.958} C_VEL
LIN {X 0,Y 397.179,Z 802.224,A -85,B 0,C 180,E1 -11124.483,E2 -11124.483} C_VEL
LIN {X 0,Y 397.816,Z 794.503,A -85,B 0,C 180,E1 -11126.13,E2 -11126.13} C_VEL
LIN {X 0,Y 398.643,Z 785.782,A -85,B 0,C 180,E1 -11127.614,E2 -11127.614} C_VEL
LIN {X 0,Y 399.416,Z 776.606,A -85,B 0,C 180,E1 -11128.878,E2 -11128.878} C_VEL
LIN {X 0,Y 400.298,Z 765.296,A -85,B 0,C 180,E1 -11130.121,E2 -11130.121} C_VEL
LIN {X 0,Y 401.193,Z 753.403,A -85,B 0,C 180,E1 -11131.147,E2 -11131.147} C_VEL
LIN {X 0,Y 401.936,Z 740.89,A -85,B 0,C 180,E1 -11131.967,E2 -11131.967} C_VEL
LIN {X 0,Y 402.435,Z 728.068,A -85,B 0,C 180,E1 -11132.587,E2 -11132.587} C_VEL
LIN {X 0,Y 402.843,Z 715.072,A -85,B 0,C 180,E1 -11132.991,E2 -11132.991} C_VEL
LIN {X 0,Y 404.275,Z 630.62,A -85,B 0,C 180,E1 -11134.62,E2 -11134.62} C_VEL
LIN {X 0,Y 400.691,Z 615.238,A -85,B 0,C 180,E1 -11135.141,E2 -11135.141} C_VEL
LIN {X 0,Y 399.145,Z 610.959,A -85,B 0,C 180,E1 -11135.35,E2 -11135.35} C_VEL
LIN {X 0,Y 397.136,Z 601.018,A -85,B 0,C 180,E1 -11138.253,E2 -11138.253} C_VEL
LIN {X 0,Y 397.152,Z 601.014,A -85,B 0,C 180,E1 -11141.427,E2 -11141.427} C_VEL
LIN {X 0,Y 397.171,Z 601.015,A -85,B 0,C 180,E1 -11144.608,E2 -11144.608} C_VEL
LIN {X 0,Y 397.221,Z 601.004,A -85,B 0,C 180,E1 -11147.743,E2 -11147.743} C_VEL
LIN {X 0,Y 397.386,Z 600.985,A -85,B 0,C 180,E1 -11152.041,E2 -11152.041} C_VEL
LIN {X 0,Y 397.255,Z 601.004,A -85,B 0,C 180,E1 -11154.926,E2 -11154.926} C_VEL
LIN {X 0,Y 397.444,Z 600.976,A -85,B 0,C 180,E1 -11157.974,E2 -11157.974} C_VEL
LIN {X 0,Y 397.573,Z 600.96,A -85,B 0,C 180,E1 -11160.001,E2 -11160.001} C_VEL
LIN {X 0,Y 397.375,Z 600.986,A -85,B 0,C 180,E1 -11163.042,E2 -11163.042} C_VEL
LIN {X 0,Y 397.38,Z 600.983,A -85,B 0,C 180,E1 -11166.092,E2 -11166.092} C_VEL
LIN {X 0,Y 397.369,Z 600.985,A -85,B 0,C 180,E1 -11168.135,E2 -11168.135} C_VEL
LIN {X 0,Y 397.222,Z 601.002,A -85,B 0,C 180,E1 -11172.259,E2 -11172.259} C_VEL
LIN {X 0,Y 397.172,Z 601.007,A -85,B 0,C 180,E1 -11175.393,E2 -11175.393} C_VEL
LIN {X 0,Y 397.155,Z 601.012,A -85,B 0,C 180,E1 -11178.574,E2 -11178.574} C_VEL
LIN {X 0,Y 397.089,Z 601.017,A -85,B 0,C 180,E1 -11181.819,E2 -11181.819} C_VEL
LIN {X 0,Y 397.15,Z 601.012,A -85,B 0,C 180,E1 -11185.133,E2 -11185.133} C_VEL
LIN {X 0,Y 397.158,Z 601.009,A -85,B 0,C 180,E1 -11187.777,E2 -11187.777} C_VEL
LIN {X 0,Y 397.083,Z 601.02,A -85,B 0,C 180,E1 -11190.883,E2 -11190.883} C_VEL
LIN {X 0,Y 397.121,Z 601.012,A -85,B 0,C 180,E1 -11194.494,E2 -11194.494} C_VEL
LIN {X 0,Y 397.104,Z 601.015,A -85,B 0,C 180,E1 -11198.275,E2 -11198.275} C_VEL
LIN {X 0,Y 397.108,Z 601.016,A -85,B 0,C 180,E1 -11200.907,E2 -11200.907} C_VEL
LIN {X 0,Y 397.102,Z 601.02,A -85,B 0,C 180,E1 -11203.649,E2 -11203.649} C_VEL
LIN {X 0,Y 397.102,Z 601.019,A -85,B 0,C 180,E1 -11206.522,E2 -11206.522} C_VEL
LIN {X 0,Y 397.119,Z 601.02,A -85,B 0,C 180,E1 -11209.552,E2 -11209.552} C_VEL
LIN {X 0,Y 397.098,Z 601.021,A -85,B 0,C 180,E1 -11212.791,E2 -11212.791} C_VEL
LIN {X 0,Y 397.118,Z 601.022,A -85,B 0,C 180,E1 -11216.283,E2 -11216.283} C_VEL
LIN {X 0,Y 397.135,Z 601.016,A -85,B 0,C 180,E1 -11220.265,E2 -11220.265} C_VEL
LIN {X 0,Y 399.723,Z 612.602,A -85,B 0,C 180,E1 -11223.055,E2 -11223.055} C_VEL
LIN {X 0,Y 401.023,Z 620.572,A -85,B 0,C 180,E1 -11224.851,E2 -11224.851} C_VEL
LIN {X 0,Y 399.561,Z 637.559,A -85,B 0,C 180,E1 -11228.323,E2 -11228.323} C_VEL
LIN {X 0,Y 399.096,Z 644.312,A -85,B 0,C 180,E1 -11229.687,E2 -11229.687} C_VEL
LIN {X 0,Y 403.258,Z 671.119,A -85,B 0,C 180,E1 -11230.472,E2 -11230.472} C_VEL
LIN {X 0,Y 403.745,Z 677.365,A -85,B 0,C 180,E1 -11230.625,E2 -11230.625} C_VEL
LIN {X 0,Y 402.539,Z 753.912,A -85,B 0,C 180,E1 -11232.112,E2 -11232.112} C_VEL
LIN {X 0,Y 401.888,Z 767.519,A -85,B 0,C 180,E1 -11232.575,E2 -11232.575} C_VEL
LIN {X 0,Y 401.128,Z 779.899,A -85,B 0,C 180,E1 -11233.197,E2 -11233.197} C_VEL
LIN {X 0,Y 400.227,Z 792.614,A -85,B 0,C 180,E1 -11234.076,E2 -11234.076} C_VEL
LIN {X 0,Y 399.348,Z 803.963,A -85,B 0,C 180,E1 -11235.086,E2 -11235.086} C_VEL
LIN {X 0,Y 398.572,Z 813.67,A -85,B 0,C 180,E1 -11236.159,E2 -11236.159} C_VEL
LIN {X 0,Y 397.78,Z 823.472,A -85,B 0,C 180,E1 -11237.501,E2 -11237.501} C_VEL
LIN {X 0,Y 396.948,Z 832.508,A -85,B 0,C 180,E1 -11239.028,E2 -11239.028} C_VEL
LIN {X 0,Y 396.459,Z 839.79,A -85,B 0,C 180,E1 -11240.563,E2 -11240.563} C_VEL
LIN {X 0,Y 396.169,Z 844.718,A -85,B 0,C 180,E1 -11241.841,E2 -11241.841} C_VEL
LIN {X 0,Y 395.967,Z 849.513,A -85,B 0,C 180,E1 -11243.376,E2 -11243.376} C_VEL
LIN {X 0,Y 395.874,Z 853.175,A -85,B 0,C 180,E1 -11244.908,E2 -11244.908} C_VEL
LIN {X 0,Y 395.804,Z 855.053,A -85,B 0,C 180,E1 -11245.927,E2 -11245.927} C_VEL
LIN {X 0,Y 395.862,Z 857.49,A -85,B 0,C 180,E1 -11247.965,E2 -11247.965} C_VEL
LIN {X 0,Y 395.831,Z 858.106,A -85,B 0,C 180,E1 -11248.983,E2 -11248.983} C_VEL
LIN {X 0,Y 395.819,Z 858.293,A -85,B 0,C 180,E1 -11250,E2 -11250} C_VEL
LIN {X 0,Y 395.831,Z 858.056,A -85,B 0,C 180,E1 -11251.017,E2 -11251.017} C_VEL
LIN {X 0,Y 395.878,Z 857.425,A -85,B 0,C 180,E1 -11252.035,E2 -11252.035} C_VEL
LIN {X 0,Y 395.789,Z 856.388,A -85,B 0,C 180,E1 -11253.054,E2 -11253.054} C_VEL
LIN {X 0,Y 395.792,Z 854.903,A -85,B 0,C 180,E1 -11254.073,E2 -11254.073} C_VEL
LIN {X 0,Y 395.843,Z 851.307,A -85,B 0,C 180,E1 -11255.825,E2 -11255.825} C_VEL
LIN {X 0,Y 396.065,Z 846.088,A -85,B 0,C 180,E1 -11257.648,E2 -11257.648} C_VEL
LIN {X 0,Y 396.377,Z 840.356,A -85,B 0,C 180,E1 -11259.182,E2 -11259.182} C_VEL
LIN {X 0,Y 396.832,Z 833.15,A -85,B 0,C 180,E1 -11260.717,E2 -11260.717} C_VEL
LIN {X 0,Y 397.598,Z 824.178,A -85,B 0,C 180,E1 -11262.246,E2 -11262.246} C_VEL
LIN {X 0,Y 398.239,Z 815.48,A -85,B 0,C 180,E1 -11263.455,E2 -11263.455} C_VEL
LIN {X 0,Y 399.033,Z 804.738,A -85,B 0,C 180,E1 -11264.665,E2 -11264.665} C_VEL
LIN {X 0,Y 399.868,Z 793.395,A -85,B 0,C 180,E1 -11265.677,E2 -11265.677} C_VEL
LIN {X 0,Y 400.716,Z 781.674,A -85,B 0,C 180,E1 -11266.493,E2 -11266.493} C_VEL
LIN {X 0,Y 401.378,Z 769.703,A -85,B 0,C 180,E1 -11267.12,E2 -11267.12} C_VEL
LIN {X 0,Y 401.95,Z 756.666,A -85,B 0,C 180,E1 -11267.587,E2 -11267.587} C_VEL
LIN {X 0,Y 402.346,Z 735.302,A -85,B 0,C 180,E1 -11268.029,E2 -11268.029} C_VEL
LIN {X 0,Y 403.104,Z 674.821,A -85,B 0,C 180,E1 -11269.169,E2 -11269.169} C_VEL
LIN {X 0,Y 398.87,Z 645.639,A -85,B 0,C 180,E1 -11269.947,E2 -11269.947} C_VEL
LIN {X 0,Y 400.024,Z 630.28,A -85,B 0,C 180,E1 -11273.01,E2 -11273.01} C_VEL
LIN {X 0,Y 400.813,Z 619.617,A -85,B 0,C 180,E1 -11275.163,E2 -11275.163} C_VEL
LIN {X 0,Y 399.158,Z 610.136,A -85,B 0,C 180,E1 -11277.243,E2 -11277.243} C_VEL
LIN {X 0,Y 397.153,Z 601.016,A -85,B 0,C 180,E1 -11279.337,E2 -11279.337} C_VEL
LIN {X 0,Y 397.114,Z 601.016,A -85,B 0,C 180,E1 -11283.272,E2 -11283.272} C_VEL
LIN {X 0,Y 397.109,Z 601.016,A -85,B 0,C 180,E1 -11285.734,E2 -11285.734} C_VEL
LIN {X 0,Y 397.115,Z 601.014,A -85,B 0,C 180,E1 -11289.576,E2 -11289.576} C_VEL
LIN {X 0,Y 397.112,Z 601.018,A -85,B 0,C 180,E1 -11292.26,E2 -11292.26} C_VEL
LIN {X 0,Y 397.086,Z 601.02,A -85,B 0,C 180,E1 -11295.067,E2 -11295.067} C_VEL
LIN {X 0,Y 397.107,Z 601.016,A -85,B 0,C 180,E1 -11298.013,E2 -11298.013} C_VEL
LIN {X 0,Y 397.131,Z 601.015,A -85,B 0,C 180,E1 -11301.137,E2 -11301.137} C_VEL
LIN {X 0,Y 397.115,Z 601.018,A -85,B 0,C 180,E1 -11304.495,E2 -11304.495} C_VEL
LIN {X 0,Y 397.107,Z 601.015,A -85,B 0,C 180,E1 -11307.93,E2 -11307.93} C_VEL
LIN {X 0,Y 397.121,Z 601.015,A -85,B 0,C 180,E1 -11311.456,E2 -11311.456} C_VEL
LIN {X 0,Y 397.146,Z 601.012,A -85,B 0,C 180,E1 -11314.487,E2 -11314.487} C_VEL
LIN {X 0,Y 397.088,Z 601.018,A -85,B 0,C 180,E1 -11318.181,E2 -11318.181} C_VEL
LIN {X 0,Y 397.155,Z 601.013,A -85,B 0,C 180,E1 -11321.426,E2 -11321.426} C_VEL
LIN {X 0,Y 397.171,Z 601.009,A -85,B 0,C 180,E1 -11324.607,E2 -11324.607} C_VEL
LIN {X 0,Y 397.212,Z 601.004,A -85,B 0,C 180,E1 -11327.741,E2 -11327.741} C_VEL
LIN {X 0,Y 397.245,Z 601,A -85,B 0,C 180,E1 -11330.837,E2 -11330.837} C_VEL
LIN {X 0,Y 397.367,Z 600.984,A -85,B 0,C 180,E1 -11333.908,E2 -11333.908} C_VEL
LIN {X 0,Y 397.443,Z 600.975,A -85,B 0,C 180,E1 -11337.973,E2 -11337.973} C_VEL
LIN {X 0,Y 397.573,Z 600.959,A -85,B 0,C 180,E1 -11339.999,E2 -11339.999} C_VEL
LIN {X 0,Y 397.374,Z 600.984,A -85,B 0,C 180,E1 -11343.041,E2 -11343.041} C_VEL
LIN {X 0,Y 397.344,Z 600.986,A -85,B 0,C 180,E1 -11346.633,E2 -11346.633} C_VEL
LIN {X 0,Y 397.247,Z 601,A -85,B 0,C 180,E1 -11349.161,E2 -11349.161} C_VEL
LIN {X 0,Y 397.21,Z 601.004,A -85,B 0,C 180,E1 -11352.258,E2 -11352.258} C_VEL
LIN {X 0,Y 397.169,Z 601.011,A -85,B 0,C 180,E1 -11355.392,E2 -11355.392} C_VEL
LIN {X 0,Y 397.152,Z 601.01,A -85,B 0,C 180,E1 -11358.573,E2 -11358.573} C_VEL
LIN {X 0,Y 397.087,Z 601.025,A -85,B 0,C 180,E1 -11361.818,E2 -11361.818} C_VEL
LIN {X 0,Y 397.147,Z 601.011,A -85,B 0,C 180,E1 -11365.132,E2 -11365.132} C_VEL
LIN {X 0,Y 397.154,Z 601.015,A -85,B 0,C 180,E1 -11367.777,E2 -11367.777} C_VEL
LIN {X 0,Y 397.077,Z 601.019,A -85,B 0,C 180,E1 -11370.882,E2 -11370.882} C_VEL
LIN {X 0,Y 397.117,Z 601.017,A -85,B 0,C 180,E1 -11374.493,E2 -11374.493} C_VEL
LIN {X 0,Y 397.102,Z 601.022,A -85,B 0,C 180,E1 -11378.274,E2 -11378.274} C_VEL
LIN {X 0,Y 397.148,Z 601.015,A -85,B 0,C 180,E1 -11381.994,E2 -11381.994} C_VEL
LIN {X 0,Y 397.106,Z 601.016,A -85,B 0,C 180,E1 -11385.065,E2 -11385.065} C_VEL
LIN {X 0,Y 397.102,Z 601.02,A -85,B 0,C 180,E1 -11388.015,E2 -11388.015} C_VEL
LIN {X 0,Y 397.127,Z 601.013,A -85,B 0,C 180,E1 -11391.138,E2 -11391.138} C_VEL
LIN {X 0,Y 397.114,Z 601.021,A -85,B 0,C 180,E1 -11394.497,E2 -11394.497} C_VEL
LIN {X 0,Y 397.072,Z 601.021,A -85,B 0,C 180,E1 -11397.929,E2 -11397.929} C_VEL
LIN {X 0,Y 397.116,Z 601.014,A -85,B 0,C 180,E1 -11401.457,E2 -11401.457} C_VEL
LIN {X 0,Y 397.148,Z 601.016,A -85,B 0,C 180,E1 -11404.488,E2 -11404.488} C_VEL
LIN {X 0,Y 397.104,Z 601.017,A -85,B 0,C 180,E1 -11408.183,E2 -11408.183} C_VEL
LIN {X 0,Y 397.158,Z 601.01,A -85,B 0,C 180,E1 -11411.427,E2 -11411.427} C_VEL
LIN {X 0,Y 397.177,Z 601.012,A -85,B 0,C 180,E1 -11414.608,E2 -11414.608} C_VEL
LIN {X 0,Y 397.216,Z 601.002,A -85,B 0,C 180,E1 -11417.742,E2 -11417.742} C_VEL
LIN {X 0,Y 397.25,Z 601.004,A -85,B 0,C 180,E1 -11420.838,E2 -11420.838} C_VEL
LIN {X 0,Y 397.367,Z 600.983,A -85,B 0,C 180,E1 -11423.909,E2 -11423.909} C_VEL
LIN {X 0,Y 397.449,Z 600.973,A -85,B 0,C 180,E1 -11427.973,E2 -11427.973} C_VEL
LIN {X 0,Y 397.578,Z 600.957,A -85,B 0,C 180,E1 -11430,E2 -11430} C_VEL
LIN {X 0,Y 397.379,Z 600.988,A -85,B 0,C 180,E1 -11433.041,E2 -11433.041} C_VEL
LIN {X 0,Y 397.367,Z 600.983,A -85,B 0,C 180,E1 -11436.091,E2 -11436.091} C_VEL
LIN {X 0,Y 397.25,Z 601.004,A -85,B 0,C 180,E1 -11439.162,E2 -11439.162} C_VEL
LIN {X 0,Y 397.216,Z 601.002,A -85,B 0,C 180,E1 -11442.258,E2 -11442.258} C_VEL
LIN {X 0,Y 397.176,Z 601.014,A -85,B 0,C 180,E1 -11445.392,E2 -11445.392} C_VEL
LIN {X 0,Y 397.158,Z 601.01,A -85,B 0,C 180,E1 -11448.573,E2 -11448.573} C_VEL
LIN {X 0,Y 397.114,Z 601.018,A -85,B 0,C 180,E1 -11451.927,E2 -11451.927} C_VEL
LIN {X 0,Y 397.162,Z 601.174,A -85,B 0,C 180,E1 -11452.842,E2 -11452.842} C_VEL
LIN {X 0,Y 398.449,Z 607.727,A -85,B 0,C 180,E1 -11454.647,E2 -11454.647} C_VEL
LIN {X 0,Y 399.314,Z 609.7,A -85,B 0,C 180,E1 -11455.007,E2 -11455.007} C_VEL
LIN {X 0,Y 400.772,Z 612.219,A -85,B 0,C 180,E1 -11455.255,E2 -11455.255} C_VEL
LIN {X 0,Y 402.415,Z 615.94,A -85,B 0,C 180,E1 -11455.443,E2 -11455.443} C_VEL
LIN {X 0,Y 402.695,Z 619.326,A -85,B 0,C 180,E1 -11455.523,E2 -11455.523} C_VEL
LIN {X 0,Y 401.363,Z 623.741,A -85,B 0,C 180,E1 -11455.546,E2 -11455.546} C_VEL
LIN {X 0,Y 398.446,Z 630.635,A -85,B 0,C 180,E1 -11455.549,E2 -11455.549} C_VEL
LIN {X 0,Y 396.731,Z 638.718,A -85,B 0,C 180,E1 -11455.629,E2 -11455.629} C_VEL
LIN {X 0,Y 395.318,Z 717.375,A -85,B 0,C 180,E1 -11457.155,E2 -11457.155} C_VEL
LIN {X 0,Y 394.914,Z 730.829,A -85,B 0,C 180,E1 -11457.633,E2 -11457.633} C_VEL
LIN {X 0,Y 394.389,Z 742.758,A -85,B 0,C 180,E1 -11458.251,E2 -11458.251} C_VEL
LIN {X 0,Y 393.716,Z 753.631,A -85,B 0,C 180,E1 -11458.995,E2 -11458.995} C_VEL
LIN {X 0,Y 392.891,Z 765.613,A -85,B 0,C 180,E1 -11460.056,E2 -11460.056} C_VEL
LIN {X 0,Y 392.107,Z 775.533,A -85,B 0,C 180,E1 -11461.154,E2 -11461.154} C_VEL
LIN {X 0,Y 391.372,Z 784.959,A -85,B 0,C 180,E1 -11462.437,E2 -11462.437} C_VEL
LIN {X 0,Y 390.629,Z 793.618,A -85,B 0,C 180,E1 -11463.898,E2 -11463.898} C_VEL
LIN {X 0,Y 389.967,Z 801.26,A -85,B 0,C 180,E1 -11465.499,E2 -11465.499} C_VEL
LIN {X 0,Y 389.565,Z 806.924,A -85,B 0,C 180,E1 -11466.981,E2 -11466.981} C_VEL
LIN {X 0,Y 389.22,Z 811.407,A -85,B 0,C 180,E1 -11468.45,E2 -11468.45} C_VEL
LIN {X 0,Y 388.952,Z 814.855,A -85,B 0,C 180,E1 -11469.899,E2 -11469.899} C_VEL
LIN {X 0,Y 388.72,Z 818.296,A -85,B 0,C 180,E1 -11471.985,E2 -11471.985} C_VEL
LIN {X 0,Y 388.607,Z 819.815,A -85,B 0,C 180,E1 -11473.665,E2 -11473.665} C_VEL
LIN {X 0,Y 388.571,Z 820.293,A -85,B 0,C 180,E1 -11475.14,E2 -11475.14} C_VEL
LIN {X 0,Y 388.629,Z 819.935,A -85,B 0,C 180,E1 -11476.592,E2 -11476.592} C_VEL
LIN {X 0,Y 388.726,Z 818.832,A -85,B 0,C 180,E1 -11478.015,E2 -11478.015} C_VEL
LIN {X 0,Y 388.987,Z 815.834,A -85,B 0,C 180,E1 -11480.105,E2 -11480.105} C_VEL
LIN {X 0,Y 389.294,Z 812.694,A -85,B 0,C 180,E1 -11481.547,E2 -11481.547} C_VEL
LIN {X 0,Y 389.605,Z 808.546,A -85,B 0,C 180,E1 -11483.016,E2 -11483.016} C_VEL
LIN {X 0,Y 390.14,Z 803.244,A -85,B 0,C 180,E1 -11484.504,E2 -11484.504} C_VEL
LIN {X 0,Y 390.765,Z 796.075,A -85,B 0,C 180,E1 -11486.115,E2 -11486.115} C_VEL
LIN {X 0,Y 391.53,Z 788.232,A -85,B 0,C 180,E1 -11487.526,E2 -11487.526} C_VEL
LIN {X 0,Y 392.388,Z 779.178,A -85,B 0,C 180,E1 -11488.855,E2 -11488.855} C_VEL
LIN {X 0,Y 393.288,Z 768.7,A -85,B 0,C 180,E1 -11490.103,E2 -11490.103} C_VEL
LIN {X 0,Y 394.146,Z 757.755,A -85,B 0,C 180,E1 -11491.134,E2 -11491.134} C_VEL
LIN {X 0,Y 394.945,Z 745.889,A -85,B 0,C 180,E1 -11492.009,E2 -11492.009} C_VEL
LIN {X 0,Y 395.623,Z 732.96,A -85,B 0,C 180,E1 -11492.722,E2 -11492.722} C_VEL
LIN {X 0,Y 396.025,Z 720.846,A -85,B 0,C 180,E1 -11493.183,E2 -11493.183} C_VEL
LIN {X 0,Y 396.411,Z 702.006,A -85,B 0,C 180,E1 -11493.602,E2 -11493.602} C_VEL
LIN {X 0,Y 397.702,Z 631.628,A -85,B 0,C 180,E1 -11494.976,E2 -11494.976} C_VEL
LIN {X 0,Y 394.299,Z 617.333,A -85,B 0,C 180,E1 -11495.484,E2 -11495.484} C_VEL
LIN {X 0,Y 392.043,Z 611.452,A -85,B 0,C 180,E1 -11495.757,E2 -11495.757} C_VEL
LIN {X 0,Y 390.063,Z 601.898,A -85,B 0,C 180,E1 -11498.671,E2 -11498.671} C_VEL
LIN {X 0,Y 390.118,Z 601.893,A -85,B 0,C 180,E1 -11502.167,E2 -11502.167} C_VEL
LIN {X 0,Y 390.138,Z 601.888,A -85,B 0,C 180,E1 -11505.393,E2 -11505.393} C_VEL
LIN {X 0,Y 390.152,Z 601.889,A -85,B 0,C 180,E1 -11508.572,E2 -11508.572} C_VEL
LIN {X 0,Y 390.335,Z 601.863,A -85,B 0,C 180,E1 -11511.993,E2 -11511.993} C_VEL
LIN {X 0,Y 390.227,Z 601.878,A -85,B 0,C 180,E1 -11514.834,E2 -11514.834} C_VEL
LIN {X 0,Y 390.413,Z 601.852,A -85,B 0,C 180,E1 -11517.937,E2 -11517.937} C_VEL
LIN {X 0,Y 390.543,Z 601.836,A -85,B 0,C 180,E1 -11520.001,E2 -11520.001} C_VEL
LIN {X 0,Y 390.309,Z 601.865,A -85,B 0,C 180,E1 -11523.097,E2 -11523.097} C_VEL
LIN {X 0,Y 390.332,Z 601.861,A -85,B 0,C 180,E1 -11526.202,E2 -11526.202} C_VEL
LIN {X 0,Y 390.307,Z 601.865,A -85,B 0,C 180,E1 -11528.283,E2 -11528.283} C_VEL
LIN {X 0,Y 390.171,Z 601.882,A -85,B 0,C 180,E1 -11532.484,E2 -11532.484} C_VEL
LIN {X 0,Y 390.132,Z 601.882,A -85,B 0,C 180,E1 -11535.678,E2 -11535.678} C_VEL
LIN {X 0,Y 390.098,Z 601.891,A -85,B 0,C 180,E1 -11538.923,E2 -11538.923} C_VEL
LIN {X 0,Y 390.033,Z 601.895,A -85,B 0,C 180,E1 -11542.235,E2 -11542.235} C_VEL
LIN {X 0,Y 390.113,Z 601.885,A -85,B 0,C 180,E1 -11545.744,E2 -11545.744} C_VEL
LIN {X 0,Y 390.06,Z 601.892,A -85,B 0,C 180,E1 -11549.11,E2 -11549.11} C_VEL
LIN {X 0,Y 390.051,Z 601.891,A -85,B 0,C 180,E1 -11552.721,E2 -11552.721} C_VEL
LIN {X 0,Y 390.053,Z 601.897,A -85,B 0,C 180,E1 -11555.827,E2 -11555.827} C_VEL
LIN {X 0,Y 390.07,Z 601.896,A -85,B 0,C 180,E1 -11559.22,E2 -11559.22} C_VEL
LIN {X 0,Y 390.078,Z 601.893,A -85,B 0,C 180,E1 -11562.381,E2 -11562.381} C_VEL
LIN {X 0,Y 390.053,Z 601.898,A -85,B 0,C 180,E1 -11566.115,E2 -11566.115} C_VEL
LIN {X 0,Y 390.073,Z 601.897,A -85,B 0,C 180,E1 -11569.564,E2 -11569.564} C_VEL
LIN {X 0,Y 390.046,Z 601.899,A -85,B 0,C 180,E1 -11572.449,E2 -11572.449} C_VEL
LIN {X 0,Y 390.068,Z 601.9,A -85,B 0,C 180,E1 -11576.046,E2 -11576.046} C_VEL
LIN {X 0,Y 390.06,Z 602.009,A -85,B 0,C 180,E1 -11579.934,E2 -11579.934} C_VEL
LIN {X 0,Y 392.506,Z 612.636,A -85,B 0,C 180,E1 -11582.545,E2 -11582.545} C_VEL
LIN {X 0,Y 393.959,Z 620.439,A -85,B 0,C 180,E1 -11584.368,E2 -11584.368} C_VEL
LIN {X 0,Y 393.952,Z 624.185,A -85,B 0,C 180,E1 -11585.179,E2 -11585.179} C_VEL
LIN {X 0,Y 392.352,Z 642.624,A -85,B 0,C 180,E1 -11589.008,E2 -11589.008} C_VEL
LIN {X 0,Y 392.232,Z 643.935,A -85,B 0,C 180,E1 -11589.276,E2 -11589.276} C_VEL
LIN {X 0,Y 395.841,Z 666.174,A -85,B 0,C 180,E1 -11589.959,E2 -11589.959} C_VEL
LIN {X 0,Y 397.138,Z 676.807,A -85,B 0,C 180,E1 -11590.252,E2 -11590.252} C_VEL
LIN {X 0,Y 395.863,Z 753.323,A -85,B 0,C 180,E1 -11591.766,E2 -11591.766} C_VEL
LIN {X 0,Y 395.189,Z 766.959,A -85,B 0,C 180,E1 -11592.236,E2 -11592.236} C_VEL
LIN {X 0,Y 394.323,Z 779.888,A -85,B 0,C 180,E1 -11592.898,E2 -11592.898} C_VEL
LIN {X 0,Y 393.405,Z 792.494,A -85,B 0,C 180,E1 -11593.792,E2 -11593.792} C_VEL
LIN {X 0,Y 392.455,Z 803.779,A -85,B 0,C 180,E1 -11594.817,E2 -11594.817} C_VEL
LIN {X 0,Y 391.606,Z 813.985,A -85,B 0,C 180,E1 -11595.979,E2 -11595.979} C_VEL
LIN {X 0,Y 390.829,Z 823.226,A -85,B 0,C 180,E1 -11597.275,E2 -11597.275} C_VEL
LIN {X 0,Y 389.952,Z 832.249,A -85,B 0,C 180,E1 -11598.829,E2 -11598.829} C_VEL
LIN {X 0,Y 389.43,Z 839.512,A -85,B 0,C 180,E1 -11600.391,E2 -11600.391} C_VEL
LIN {X 0,Y 388.995,Z 846.141,A -85,B 0,C 180,E1 -11602.212,E2 -11602.212} C_VEL
LIN {X 0,Y 388.8,Z 850.654,A -85,B 0,C 180,E1 -11603.823,E2 -11603.823} C_VEL
LIN {X 0,Y 388.77,Z 852.869,A -85,B 0,C 180,E1 -11604.814,E2 -11604.814} C_VEL
LIN {X 0,Y 388.727,Z 854.734,A -85,B 0,C 180,E1 -11605.853,E2 -11605.853} C_VEL
LIN {X 0,Y 388.776,Z 857.159,A -85,B 0,C 180,E1 -11607.928,E2 -11607.928} C_VEL
LIN {X 0,Y 388.761,Z 857.771,A -85,B 0,C 180,E1 -11608.964,E2 -11608.964} C_VEL
LIN {X 0,Y 388.746,Z 857.944,A -85,B 0,C 180,E1 -11610,E2 -11610} C_VEL
LIN {X 0,Y 388.761,Z 857.701,A -85,B 0,C 180,E1 -11611.036,E2 -11611.036} C_VEL
LIN {X 0,Y 388.79,Z 857.063,A -85,B 0,C 180,E1 -11612.072,E2 -11612.072} C_VEL
LIN {X 0,Y 388.692,Z 856.017,A -85,B 0,C 180,E1 -11613.109,E2 -11613.109} C_VEL
LIN {X 0,Y 388.717,Z 854.517,A -85,B 0,C 180,E1 -11614.147,E2 -11614.147} C_VEL
LIN {X 0,Y 388.745,Z 851.276,A -85,B 0,C 180,E1 -11615.777,E2 -11615.777} C_VEL
LIN {X 0,Y 388.934,Z 847.298,A -85,B 0,C 180,E1 -11617.267,E2 -11617.267} C_VEL
LIN {X 0,Y 389.263,Z 840.924,A -85,B 0,C 180,E1 -11619.089,E2 -11619.089} C_VEL
LIN {X 0,Y 389.712,Z 833.973,A -85,B 0,C 180,E1 -11620.652,E2 -11620.652} C_VEL
LIN {X 0,Y 390.468,Z 825.277,A -85,B 0,C 180,E1 -11622.209,E2 -11622.209} C_VEL
LIN {X 0,Y 391.277,Z 815.114,A -85,B 0,C 180,E1 -11623.667,E2 -11623.667} C_VEL
LIN {X 0,Y 392.019,Z 805.335,A -85,B 0,C 180,E1 -11624.801,E2 -11624.801} C_VEL
LIN {X 0,Y 392.869,Z 794.216,A -85,B 0,C 180,E1 -11625.831,E2 -11625.831} C_VEL
LIN {X 0,Y 393.81,Z 781.793,A -85,B 0,C 180,E1 -11626.724,E2 -11626.724} C_VEL
LIN {X 0,Y 394.507,Z 770.023,A -85,B 0,C 180,E1 -11627.361,E2 -11627.361} C_VEL
LIN {X 0,Y 395.074,Z 757.359,A -85,B 0,C 180,E1 -11627.836,E2 -11627.836} C_VEL
LIN {X 0,Y 395.46,Z 738.262,A -85,B 0,C 180,E1 -11628.253,E2 -11628.253} C_VEL
LIN {X 0,Y 396.321,Z 675.435,A -85,B 0,C 180,E1 -11629.46,E2 -11629.46} C_VEL
LIN {X 0,Y 391.959,Z 645.268,A -85,B 0,C 180,E1 -11630.294,E2 -11630.294} C_VEL
LIN {X 0,Y 393.413,Z 627.175,A -85,B 0,C 180,E1 -11633.979,E2 -11633.979} C_VEL
LIN {X 0,Y 393.845,Z 620.511,A -85,B 0,C 180,E1 -11635.357,E2 -11635.357} C_VEL
LIN {X 0,Y 391.785,Z 609.638,A -85,B 0,C 180,E1 -11637.8,E2 -11637.8} C_VEL
LIN {X 0,Y 390.103,Z 601.893,A -85,B 0,C 180,E1 -11639.623,E2 -11639.623} C_VEL
LIN {X 0,Y 390.043,Z 601.902,A -85,B 0,C 180,E1 -11642.721,E2 -11642.721} C_VEL
LIN {X 0,Y 390.057,Z 601.894,A -85,B 0,C 180,E1 -11645.825,E2 -11645.825} C_VEL
LIN {X 0,Y 390.073,Z 601.892,A -85,B 0,C 180,E1 -11649.218,E2 -11649.218} C_VEL
LIN {X 0,Y 390.078,Z 601.896,A -85,B 0,C 180,E1 -11652.379,E2 -11652.379} C_VEL
LIN {X 0,Y 390.055,Z 601.895,A -85,B 0,C 180,E1 -11656.112,E2 -11656.112} C_VEL
LIN {X 0,Y 390.07,Z 601.892,A -85,B 0,C 180,E1 -11659.562,E2 -11659.562} C_VEL
LIN {X 0,Y 390.055,Z 601.897,A -85,B 0,C 180,E1 -11662.445,E2 -11662.445} C_VEL
LIN {X 0,Y 390.063,Z 601.893,A -85,B 0,C 180,E1 -11666.044,E2 -11666.044} C_VEL
LIN {X 0,Y 390.044,Z 601.898,A -85,B 0,C 180,E1 -11668.497,E2 -11668.497} C_VEL
LIN {X 0,Y 390.112,Z 601.887,A -85,B 0,C 180,E1 -11672.069,E2 -11672.069} C_VEL
LIN {X 0,Y 390.071,Z 601.894,A -85,B 0,C 180,E1 -11675.518,E2 -11675.518} C_VEL
LIN {X 0,Y 390.048,Z 601.899,A -85,B 0,C 180,E1 -11678.877,E2 -11678.877} C_VEL
LIN {X 0,Y 390.121,Z 601.885,A -85,B 0,C 180,E1 -11682.166,E2 -11682.166} C_VEL
LIN {X 0,Y 390.135,Z 601.889,A -85,B 0,C 180,E1 -11685.392,E2 -11685.392} C_VEL
LIN {X 0,Y 390.141,Z 601.884,A -85,B 0,C 180,E1 -11688.57,E2 -11688.57} C_VEL
LIN {X 0,Y 390.299,Z 601.864,A -85,B 0,C 180,E1 -11692.031,E2 -11692.031} C_VEL
LIN {X 0,Y 390.221,Z 601.875,A -85,B 0,C 180,E1 -11694.833,E2 -11694.833} C_VEL
LIN {X 0,Y 390.412,Z 601.851,A -85,B 0,C 180,E1 -11697.936,E2 -11697.936} C_VEL
LIN {X 0,Y 390.543,Z 601.835,A -85,B 0,C 180,E1 -11699.999,E2 -11699.999} C_VEL
LIN {X 0,Y 390.309,Z 601.865,A -85,B 0,C 180,E1 -11703.096,E2 -11703.096} C_VEL
LIN {X 0,Y 390.299,Z 601.863,A -85,B 0,C 180,E1 -11706.627,E2 -11706.627} C_VEL
LIN {X 0,Y 390.199,Z 601.88,A -85,B 0,C 180,E1 -11709.328,E2 -11709.328} C_VEL
LIN {X 0,Y 390.185,Z 601.882,A -85,B 0,C 180,E1 -11713.438,E2 -11713.438} C_VEL
LIN {X 0,Y 390.139,Z 601.885,A -85,B 0,C 180,E1 -11717.307,E2 -11717.307} C_VEL
LIN {X 0,Y 390.078,Z 601.892,A -85,B 0,C 180,E1 -11720.47,E2 -11720.47} C_VEL
LIN {X 0,Y 390.08,Z 601.892,A -85,B 0,C 180,E1 -11723.351,E2 -11723.351} C_VEL
LIN {X 0,Y 390.104,Z 601.888,A -85,B 0,C 180,E1 -11726.768,E2 -11726.768} C_VEL
LIN {X 0,Y 390.036,Z 601.9,A -85,B 0,C 180,E1 -11730.299,E2 -11730.299} C_VEL
LIN {X 0,Y 390.076,Z 601.897,A -85,B 0,C 180,E1 -11733.953,E2 -11733.953} C_VEL
LIN {X 0,Y 390.039,Z 601.897,A -85,B 0,C 180,E1 -11737.552,E2 -11737.552} C_VEL
LIN {X 0,Y 390.075,Z 601.892,A -85,B 0,C 180,E1 -11740.826,E2 -11740.826} C_VEL
LIN {X 0,Y 390.097,Z 601.892,A -85,B 0,C 180,E1 -11743.894,E2 -11743.894} C_VEL
LIN {X 0,Y 390.074,Z 601.892,A -85,B 0,C 180,E1 -11747.62,E2 -11747.62} C_VEL
LIN {X 0,Y 390.086,Z 601.892,A -85,B 0,C 180,E1 -11750.908,E2 -11750.908} C_VEL
LIN {X 0,Y 390.079,Z 601.894,A -85,B 0,C 180,E1 -11754.794,E2 -11754.794} C_VEL
LIN {X 0,Y 390.018,Z 601.906,A -85,B 0,C 180,E1 -11758.496,E2 -11758.496} C_VEL
LIN {X 0,Y 390.112,Z 601.888,A -85,B 0,C 180,E1 -11762.07,E2 -11762.07} C_VEL
LIN {X 0,Y 390.075,Z 601.891,A -85,B 0,C 180,E1 -11765.52,E2 -11765.52} C_VEL
LIN {X 0,Y 390.058,Z 601.898,A -85,B 0,C 180,E1 -11768.878,E2 -11768.878} C_VEL
LIN {X 0,Y 390.124,Z 601.886,A -85,B 0,C 180,E1 -11772.167,E2 -11772.167} C_VEL
LIN {X 0,Y 390.143,Z 601.884,A -85,B 0,C 180,E1 -11775.393,E2 -11775.393} C_VEL
LIN {X 0,Y 390.145,Z 601.886,A -85,B 0,C 180,E1 -11778.571,E2 -11778.571} C_VEL
LIN {X 0,Y 390.304,Z 601.863,A -85,B 0,C 180,E1 -11782.032,E2 -11782.032} C_VEL
LIN {X 0,Y 390.223,Z 601.878,A -85,B 0,C 180,E1 -11784.834,E2 -11784.834} C_VEL
LIN {X 0,Y 390.418,Z 601.849,A -85,B 0,C 180,E1 -11787.937,E2 -11787.937} C_VEL
LIN {X 0,Y 390.547,Z 601.832,A -85,B 0,C 180,E1 -11790,E2 -11790} C_VEL
LIN {X 0,Y 390.313,Z 601.869,A -85,B 0,C 180,E1 -11793.096,E2 -11793.096} C_VEL
LIN {X 0,Y 390.321,Z 601.861,A -85,B 0,C 180,E1 -11796.202,E2 -11796.202} C_VEL
LIN {X 0,Y 390.202,Z 601.882,A -85,B 0,C 180,E1 -11799.329,E2 -11799.329} C_VEL
LIN {X 0,Y 390.167,Z 601.88,A -85,B 0,C 180,E1 -11802.483,E2 -11802.483} C_VEL
LIN {X 0,Y 390.136,Z 601.887,A -85,B 0,C 180,E1 -11805.677,E2 -11805.677} C_VEL
LIN {X 0,Y 390.102,Z 601.89,A -85,B 0,C 180,E1 -11808.922,E2 -11808.922} C_VEL
LIN {X 0,Y 390.106,Z 601.931,A -85,B 0,C 180,E1 -11812.578,E2 -11812.578} C_VEL
LIN {X 0,Y 391.669,Z 610.051,A -85,B 0,C 180,E1 -11814.798,E2 -11814.798} C_VEL
LIN {X 0,Y 394.111,Z 618.44,A -85,B 0,C 180,E1 -11815.092,E2 -11815.092} C_VEL
LIN {X 0,Y 396.871,Z 631.996,A -85,B 0,C 180,E1 -11815.501,E2 -11815.501} C_VEL
LIN {X 0,Y 396.731,Z 638.718,A -85,B 0,C 180,E1 -11815.629,E2 -11815.629} C_VEL
LIN {X 0,Y 395.926,Z 644.551,A -85,B 0,C 180,E1 -11815.707,E2 -11815.707} C_VEL
LIN {X 0,Y 390.191,Z 663.516,A -85,B 0,C 180,E1 -11815.819,E2 -11815.819} C_VEL
LIN {X 0,Y 389.394,Z 669.348,A -85,B 0,C 180,E1 -11815.901,E2 -11815.901} C_VEL
LIN {X 0,Y 388.521,Z 717.741,A -85,B 0,C 180,E1 -11816.868,E2 -11816.868} C_VEL
LIN {X 0,Y 388.094,Z 731.591,A -85,B 0,C 180,E1 -11817.373,E2 -11817.373} C_VEL
LIN {X 0,Y 387.507,Z 744.002,A -85,B 0,C 180,E1 -11818.04,E2 -11818.04} C_VEL
LIN {X 0,Y 386.699,Z 756.38,A -85,B 0,C 180,E1 -11818.939,E2 -11818.939} C_VEL
LIN {X 0,Y 385.919,Z 766.775,A -85,B 0,C 180,E1 -11819.902,E2 -11819.902} C_VEL
LIN {X 0,Y 385.049,Z 777.576,A -85,B 0,C 180,E1 -11821.151,E2 -11821.151} C_VEL
LIN {X 0,Y 384.273,Z 787.07,A -85,B 0,C 180,E1 -11822.526,E2 -11822.526} C_VEL
LIN {X 0,Y 383.435,Z 796.057,A -85,B 0,C 180,E1 -11824.134,E2 -11824.134} C_VEL
LIN {X 0,Y 382.855,Z 802.808,A -85,B 0,C 180,E1 -11825.649,E2 -11825.649} C_VEL
LIN {X 0,Y 382.404,Z 808.779,A -85,B 0,C 180,E1 -11827.335,E2 -11827.335} C_VEL
LIN {X 0,Y 382.109,Z 812.654,A -85,B 0,C 180,E1 -11828.707,E2 -11828.707} C_VEL
LIN {X 0,Y 381.843,Z 815.75,A -85,B 0,C 180,E1 -11830.104,E2 -11830.104} C_VEL
LIN {X 0,Y 381.67,Z 818.06,A -85,B 0,C 180,E1 -11831.52,E2 -11831.52} C_VEL
LIN {X 0,Y 381.574,Z 819.647,A -85,B 0,C 180,E1 -11832.958,E2 -11832.958} C_VEL
LIN {X 0,Y 381.478,Z 820.509,A -85,B 0,C 180,E1 -11834.432,E2 -11834.432} C_VEL
LIN {X 0,Y 381.489,Z 820.559,A -85,B 0,C 180,E1 -11835.928,E2 -11835.928} C_VEL
LIN {X 0,Y 381.607,Z 819.771,A -85,B 0,C 180,E1 -11837.447,E2 -11837.447} C_VEL
LIN {X 0,Y 381.732,Z 818.095,A -85,B 0,C 180,E1 -11839.01,E2 -11839.01} C_VEL
LIN {X 0,Y 382.023,Z 815.454,A -85,B 0,C 180,E1 -11840.592,E2 -11840.592} C_VEL
LIN {X 0,Y 382.365,Z 811.692,A -85,B 0,C 180,E1 -11842.217,E2 -11842.217} C_VEL
LIN {X 0,Y 382.861,Z 806.127,A -85,B 0,C 180,E1 -11844.027,E2 -11844.027} C_VEL
LIN {X 0,Y 383.445,Z 800.07,A -85,B 0,C 180,E1 -11845.565,E2 -11845.565} C_VEL
LIN {X 0,Y 384.172,Z 792.915,A -85,B 0,C 180,E1 -11847.029,E2 -11847.029} C_VEL
LIN {X 0,Y 385.16,Z 783.646,A -85,B 0,C 180,E1 -11848.554,E2 -11848.554} C_VEL
LIN {X 0,Y 386.017,Z 774.287,A -85,B 0,C 180,E1 -11849.805,E2 -11849.805} C_VEL
LIN {X 0,Y 386.93,Z 763.861,A -85,B 0,C 180,E1 -11850.931,E2 -11850.931} C_VEL
LIN {X 0,Y 387.801,Z 752.638,A -85,B 0,C 180,E1 -11851.889,E2 -11851.889} C_VEL
LIN {X 0,Y 388.61,Z 740.325,A -85,B 0,C 180,E1 -11852.699,E2 -11852.699} C_VEL
LIN {X 0,Y 389.087,Z 727.442,A -85,B 0,C 180,E1 -11853.319,E2 -11853.319} C_VEL
LIN {X 0,Y 389.564,Z 714.296,A -85,B 0,C 180,E1 -11853.716,E2 -11853.716} C_VEL
LIN {X 0,Y 391.068,Z 632.335,A -85,B 0,C 180,E1 -11855.363,E2 -11855.363} C_VEL
LIN {X 0,Y 388.117,Z 619.966,A -85,B 0,C 180,E1 -11855.816,E2 -11855.816} C_VEL
LIN {X 0,Y 384.891,Z 611.792,A -85,B 0,C 180,E1 -11856.23,E2 -11856.23} C_VEL
LIN {X 0,Y 383.025,Z 602.777,A -85,B 0,C 180,E1 -11859.02,E2 -11859.02} C_VEL
LIN {X 0,Y 383.085,Z 602.769,A -85,B 0,C 180,E1 -11862.546,E2 -11862.546} C_VEL
LIN {X 0,Y 383.117,Z 602.764,A -85,B 0,C 180,E1 -11866.464,E2 -11866.464} C_VEL
LIN {X 0,Y 383.133,Z 602.761,A -85,B 0,C 180,E1 -11869.431,E2 -11869.431} C_VEL
LIN {X 0,Y 383.265,Z 602.745,A -85,B 0,C 180,E1 -11872.626,E2 -11872.626} C_VEL
LIN {X 0,Y 383.198,Z 602.753,A -85,B 0,C 180,E1 -11874.739,E2 -11874.739} C_VEL
LIN {X 0,Y 383.382,Z 602.728,A -85,B 0,C 180,E1 -11877.899,E2 -11877.899} C_VEL
LIN {X 0,Y 383.512,Z 602.711,A -85,B 0,C 180,E1 -11880.001,E2 -11880.001} C_VEL
LIN {X 0,Y 383.246,Z 602.745,A -85,B 0,C 180,E1 -11883.154,E2 -11883.154} C_VEL
LIN {X 0,Y 383.288,Z 602.739,A -85,B 0,C 180,E1 -11886.317,E2 -11886.317} C_VEL
LIN {X 0,Y 383.253,Z 602.745,A -85,B 0,C 180,E1 -11888.436,E2 -11888.436} C_VEL
LIN {X 0,Y 383.1,Z 602.762,A -85,B 0,C 180,E1 -11891.643,E2 -11891.643} C_VEL
LIN {X 0,Y 383.105,Z 602.766,A -85,B 0,C 180,E1 -11894.882,E2 -11894.882} C_VEL
LIN {X 0,Y 383.056,Z 602.767,A -85,B 0,C 180,E1 -11898.174,E2 -11898.174} C_VEL
LIN {X 0,Y 382.986,Z 602.776,A -85,B 0,C 180,E1 -11901.532,E2 -11901.532} C_VEL
LIN {X 0,Y 383.046,Z 602.771,A -85,B 0,C 180,E1 -11904.961,E2 -11904.961} C_VEL
LIN {X 0,Y 383.044,Z 602.766,A -85,B 0,C 180,E1 -11908.493,E2 -11908.493} C_VEL
LIN {X 0,Y 383.032,Z 602.764,A -85,B 0,C 180,E1 -11912.148,E2 -11912.148} C_VEL
LIN {X 0,Y 383.022,Z 602.772,A -85,B 0,C 180,E1 -11915.956,E2 -11915.956} C_VEL
LIN {X 0,Y 383.017,Z 602.775,A -85,B 0,C 180,E1 -11919.589,E2 -11919.589} C_VEL
LIN {X 0,Y 383.029,Z 602.773,A -85,B 0,C 180,E1 -11922.784,E2 -11922.784} C_VEL
LIN {X 0,Y 382.996,Z 602.777,A -85,B 0,C 180,E1 -11925.79,E2 -11925.79} C_VEL
LIN {X 0,Y 383.013,Z 602.775,A -85,B 0,C 180,E1 -11928.792,E2 -11928.792} C_VEL
LIN {X 0,Y 383.002,Z 602.778,A -85,B 0,C 180,E1 -11932.097,E2 -11932.097} C_VEL
LIN {X 0,Y 383.018,Z 602.778,A -85,B 0,C 180,E1 -11935.333,E2 -11935.333} C_VEL
LIN {X 0,Y 382.983,Z 602.778,A -85,B 0,C 180,E1 -11939.082,E2 -11939.082} C_VEL
LIN {X 0,Y 382.981,Z 602.795,A -85,B 0,C 180,E1 -11939.501,E2 -11939.501} C_VEL
LIN {X 0,Y 385.583,Z 613.883,A -85,B 0,C 180,E1 -11942.304,E2 -11942.304} C_VEL
LIN {X 0,Y 387.198,Z 622.935,A -85,B 0,C 180,E1 -11944.465,E2 -11944.465} C_VEL
LIN {X 0,Y 386.166,Z 634.645,A -85,B 0,C 180,E1 -11946.966,E2 -11946.966} C_VEL
LIN {X 0,Y 385.415,Z 643.544,A -85,B 0,C 180,E1 -11948.842,E2 -11948.842} C_VEL
LIN {X 0,Y 388.874,Z 664.404,A -85,B 0,C 180,E1 -11949.512,E2 -11949.512} C_VEL
LIN {X 0,Y 390.461,Z 676.477,A -85,B 0,C 180,E1 -11949.865,E2 -11949.865} C_VEL
LIN {X 0,Y 389.2,Z 752.789,A -85,B 0,C 180,E1 -11951.408,E2 -11951.408} C_VEL
LIN {X 0,Y 388.454,Z 766.466,A -85,B 0,C 180,E1 -11951.883,E2 -11951.883} C_VEL
LIN {X 0,Y 387.618,Z 778.9,A -85,B 0,C 180,E1 -11952.525,E2 -11952.525} C_VEL
LIN {X 0,Y 386.747,Z 790.865,A -85,B 0,C 180,E1 -11953.369,E2 -11953.369} C_VEL
LIN {X 0,Y 385.676,Z 802.378,A -85,B 0,C 180,E1 -11954.409,E2 -11954.409} C_VEL
LIN {X 0,Y 384.746,Z 813.404,A -85,B 0,C 180,E1 -11955.668,E2 -11955.668} C_VEL
LIN {X 0,Y 383.882,Z 823.009,A -85,B 0,C 180,E1 -11957.04,E2 -11957.04} C_VEL
LIN {X 0,Y 382.938,Z 831.998,A -85,B 0,C 180,E1 -11958.622,E2 -11958.622} C_VEL
LIN {X 0,Y 382.378,Z 839.232,A -85,B 0,C 180,E1 -11960.212,E2 -11960.212} C_VEL
LIN {X 0,Y 382.049,Z 844.151,A -85,B 0,C 180,E1 -11961.538,E2 -11961.538} C_VEL
LIN {X 0,Y 381.801,Z 848.922,A -85,B 0,C 180,E1 -11963.128,E2 -11963.128} C_VEL
LIN {X 0,Y 381.669,Z 852.563,A -85,B 0,C 180,E1 -11964.717,E2 -11964.717} C_VEL
LIN {X 0,Y 381.652,Z 854.416,A -85,B 0,C 180,E1 -11965.776,E2 -11965.776} C_VEL
LIN {X 0,Y 381.675,Z 856.829,A -85,B 0,C 180,E1 -11967.89,E2 -11967.89} C_VEL
LIN {X 0,Y 381.692,Z 857.435,A -85,B 0,C 180,E1 -11968.945,E2 -11968.945} C_VEL
LIN {X 0,Y 381.676,Z 857.595,A -85,B 0,C 180,E1 -11970,E2 -11970} C_VEL
LIN {X 0,Y 381.693,Z 857.344,A -85,B 0,C 180,E1 -11971.055,E2 -11971.055} C_VEL
LIN {X 0,Y 381.689,Z 856.695,A -85,B 0,C 180,E1 -11972.11,E2 -11972.11} C_VEL
LIN {X 0,Y 381.599,Z 855.639,A -85,B 0,C 180,E1 -11973.167,E2 -11973.167} C_VEL
LIN {X 0,Y 381.644,Z 854.123,A -85,B 0,C 180,E1 -11974.224,E2 -11974.224} C_VEL
LIN {X 0,Y 381.696,Z 850.279,A -85,B 0,C 180,E1 -11976.128,E2 -11976.128} C_VEL
LIN {X 0,Y 381.926,Z 845.216,A -85,B 0,C 180,E1 -11977.933,E2 -11977.933} C_VEL
LIN {X 0,Y 382.374,Z 838.289,A -85,B 0,C 180,E1 -11979.788,E2 -11979.788} C_VEL
LIN {X 0,Y 382.922,Z 830.754,A -85,B 0,C 180,E1 -11981.379,E2 -11981.379} C_VEL
LIN {X 0,Y 383.625,Z 823.073,A -85,B 0,C 180,E1 -11982.699,E2 -11982.699} C_VEL
LIN {X 0,Y 384.353,Z 814.212,A -85,B 0,C 180,E1 -11983.959,E2 -11983.959} C_VEL
LIN {X 0,Y 385.201,Z 803.358,A -85,B 0,C 180,E1 -11985.205,E2 -11985.205} C_VEL
LIN {X 0,Y 386.137,Z 791.86,A -85,B 0,C 180,E1 -11986.25,E2 -11986.25} C_VEL
LIN {X 0,Y 387.023,Z 779.884,A -85,B 0,C 180,E1 -11987.094,E2 -11987.094} C_VEL
LIN {X 0,Y 387.809,Z 766.646,A -85,B 0,C 180,E1 -11987.773,E2 -11987.773} C_VEL
LIN {X 0,Y 388.353,Z 753.608,A -85,B 0,C 180,E1 -11988.224,E2 -11988.224} C_VEL
LIN {X 0,Y 389.596,Z 676.383,A -85,B 0,C 180,E1 -11989.753,E2 -11989.753} C_VEL
LIN {X 0,Y 385.047,Z 644.98,A -85,B 0,C 180,E1 -11990.639,E2 -11990.639} C_VEL
LIN {X 0,Y 386.655,Z 626.229,A -85,B 0,C 180,E1 -11994.527,E2 -11994.527} C_VEL
LIN {X 0,Y 386.829,Z 621.356,A -85,B 0,C 180,E1 -11995.562,E2 -11995.562} C_VEL
LIN {X 0,Y 384.732,Z 610.493,A -85,B 0,C 180,E1 -11998.058,E2 -11998.058} C_VEL
LIN {X 0,Y 383.042,Z 602.772,A -85,B 0,C 180,E1 -11999.931,E2 -11999.931} C_VEL
LIN {X 0,Y 383.003,Z 602.774,A -85,B 0,C 180,E1 -12003.4,E2 -12003.4} C_VEL
LIN {X 0,Y 383.033,Z 602.772,A -85,B 0,C 180,E1 -12006.164,E2 -12006.164} C_VEL
LIN {X 0,Y 383.017,Z 602.772,A -85,B 0,C 180,E1 -12009.956,E2 -12009.956} C_VEL
LIN {X 0,Y 383.03,Z 602.774,A -85,B 0,C 180,E1 -12012.782,E2 -12012.782} C_VEL
LIN {X 0,Y 382.997,Z 602.773,A -85,B 0,C 180,E1 -12015.789,E2 -12015.789} C_VEL
LIN {X 0,Y 383.012,Z 602.777,A -85,B 0,C 180,E1 -12018.79,E2 -12018.79} C_VEL
LIN {X 0,Y 383.005,Z 602.773,A -85,B 0,C 180,E1 -12022.093,E2 -12022.093} C_VEL
LIN {X 0,Y 383.014,Z 602.773,A -85,B 0,C 180,E1 -12025.331,E2 -12025.331} C_VEL
LIN {X 0,Y 383.032,Z 602.769,A -85,B 0,C 180,E1 -12027.852,E2 -12027.852} C_VEL
LIN {X 0,Y 383.058,Z 602.766,A -85,B 0,C 180,E1 -12031.719,E2 -12031.719} C_VEL
LIN {X 0,Y 383.044,Z 602.774,A -85,B 0,C 180,E1 -12035.039,E2 -12035.039} C_VEL
LIN {X 0,Y 382.985,Z 602.776,A -85,B 0,C 180,E1 -12038.468,E2 -12038.468} C_VEL
LIN {X 0,Y 383.056,Z 602.766,A -85,B 0,C 180,E1 -12041.826,E2 -12041.826} C_VEL
LIN {X 0,Y 383.102,Z 602.766,A -85,B 0,C 180,E1 -12045.117,E2 -12045.117} C_VEL
LIN {X 0,Y 383.09,Z 602.761,A -85,B 0,C 180,E1 -12048.357,E2 -12048.357} C_VEL
LIN {X 0,Y 383.256,Z 602.742,A -85,B 0,C 180,E1 -12051.975,E2 -12051.975} C_VEL
LIN {X 0,Y 383.193,Z 602.75,A -85,B 0,C 180,E1 -12054.738,E2 -12054.738} C_VEL
LIN {X 0,Y 383.379,Z 602.727,A -85,B 0,C 180,E1 -12057.898,E2 -12057.898} C_VEL
LIN {X 0,Y 383.512,Z 602.71,A -85,B 0,C 180,E1 -12059.999,E2 -12059.999} C_VEL
LIN {X 0,Y 383.245,Z 602.745,A -85,B 0,C 180,E1 -12063.153,E2 -12063.153} C_VEL
LIN {X 0,Y 383.259,Z 602.74,A -85,B 0,C 180,E1 -12066.618,E2 -12066.618} C_VEL
LIN {X 0,Y 383.145,Z 602.76,A -85,B 0,C 180,E1 -12069.502,E2 -12069.502} C_VEL
LIN {X 0,Y 383.116,Z 602.763,A -85,B 0,C 180,E1 -12073.536,E2 -12073.536} C_VEL
LIN {X 0,Y 383.085,Z 602.766,A -85,B 0,C 180,E1 -12077.454,E2 -12077.454} C_VEL
LIN {X 0,Y 383.019,Z 602.77,A -85,B 0,C 180,E1 -12080.647,E2 -12080.647} C_VEL
LIN {X 0,Y 383.024,Z 602.776,A -85,B 0,C 180,E1 -12083.807,E2 -12083.807} C_VEL
LIN {X 0,Y 383.071,Z 602.769,A -85,B 0,C 180,E1 -12086.123,E2 -12086.123} C_VEL
LIN {X 0,Y 383.04,Z 602.769,A -85,B 0,C 180,E1 -12088.492,E2 -12088.492} C_VEL
LIN {X 0,Y 382.999,Z 602.776,A -85,B 0,C 180,E1 -12092.427,E2 -12092.427} C_VEL
LIN {X 0,Y 383.018,Z 602.776,A -85,B 0,C 180,E1 -12095.956,E2 -12095.956} C_VEL
LIN {X 0,Y 383.015,Z 602.772,A -85,B 0,C 180,E1 -12099.588,E2 -12099.588} C_VEL
LIN {X 0,Y 383.058,Z 602.767,A -85,B 0,C 180,E1 -12102.789,E2 -12102.789} C_VEL
LIN {X 0,Y 383.003,Z 602.774,A -85,B 0,C 180,E1 -12105.791,E2 -12105.791} C_VEL
LIN {X 0,Y 383.006,Z 602.774,A -85,B 0,C 180,E1 -12108.792,E2 -12108.792} C_VEL
LIN {X 0,Y 382.995,Z 602.777,A -85,B 0,C 180,E1 -12112.096,E2 -12112.096} C_VEL
LIN {X 0,Y 383.012,Z 602.771,A -85,B 0,C 180,E1 -12115.332,E2 -12115.332} C_VEL
LIN {X 0,Y 382.977,Z 602.777,A -85,B 0,C 180,E1 -12119.082,E2 -12119.082} C_VEL
LIN {X 0,Y 383.051,Z 602.772,A -85,B 0,C 180,E1 -12122.698,E2 -12122.698} C_VEL
LIN {X 0,Y 383.047,Z 602.769,A -85,B 0,C 180,E1 -12125.04,E2 -12125.04} C_VEL
LIN {X 0,Y 382.995,Z 602.778,A -85,B 0,C 180,E1 -12128.47,E2 -12128.47} C_VEL
LIN {X 0,Y 383.059,Z 602.765,A -85,B 0,C 180,E1 -12131.827,E2 -12131.827} C_VEL
LIN {X 0,Y 383.109,Z 602.763,A -85,B 0,C 180,E1 -12135.119,E2 -12135.119} C_VEL
LIN {X 0,Y 383.094,Z 602.763,A -85,B 0,C 180,E1 -12138.358,E2 -12138.358} C_VEL
LIN {X 0,Y 383.26,Z 602.74,A -85,B 0,C 180,E1 -12141.976,E2 -12141.976} C_VEL
LIN {X 0,Y 383.194,Z 602.753,A -85,B 0,C 180,E1 -12144.739,E2 -12144.739} C_VEL
LIN {X 0,Y 383.385,Z 602.725,A -85,B 0,C 180,E1 -12147.899,E2 -12147.899} C_VEL
LIN {X 0,Y 383.517,Z 602.708,A -85,B 0,C 180,E1 -12150,E2 -12150} C_VEL
LIN {X 0,Y 383.249,Z 602.749,A -85,B 0,C 180,E1 -12153.154,E2 -12153.154} C_VEL
LIN {X 0,Y 383.277,Z 602.738,A -85,B 0,C 180,E1 -12156.316,E2 -12156.316} C_VEL
LIN {X 0,Y 383.148,Z 602.758,A -85,B 0,C 180,E1 -12159.502,E2 -12159.502} C_VEL
LIN {X 0,Y 383.121,Z 602.762,A -85,B 0,C 180,E1 -12163.536,E2 -12163.536} C_VEL
LIN {X 0,Y 383.091,Z 602.768,A -85,B 0,C 180,E1 -12167.454,E2 -12167.454} C_VEL
LIN {X 0,Y 383.028,Z 602.774,A -85,B 0,C 180,E1 -12170.648,E2 -12170.648} C_VEL
LIN {X 0,Y 383.088,Z 602.922,A -85,B 0,C 180,E1 -12172.375,E2 -12172.375} C_VEL
LIN {X 0,Y 384.505,Z 610.165,A -85,B 0,C 180,E1 -12174.427,E2 -12174.427} C_VEL
LIN {X 0,Y 387.486,Z 619.987,A -85,B 0,C 180,E1 -12174.792,E2 -12174.792} C_VEL
LIN {X 0,Y 390.038,Z 632.182,A -85,B 0,C 180,E1 -12175.173,E2 -12175.173} C_VEL
LIN {X 0,Y 389.394,Z 669.348,A -85,B 0,C 180,E1 -12175.901,E2 -12175.901} C_VEL
LIN {X 0,Y 388.585,Z 675.181,A -85,B 0,C 180,E1 -12175.98,E2 -12175.98} C_VEL
LIN {X 0,Y 382.83,Z 694.142,A -85,B 0,C 180,E1 -12176.099,E2 -12176.099} C_VEL
LIN {X 0,Y 382.084,Z 699.975,A -85,B 0,C 180,E1 -12176.184,E2 -12176.184} C_VEL
LIN {X 0,Y 381.688,Z 719.924,A -85,B 0,C 180,E1 -12176.63,E2 -12176.63} C_VEL
LIN {X 0,Y 381.26,Z 733.125,A -85,B 0,C 180,E1 -12177.143,E2 -12177.143} C_VEL
LIN {X 0,Y 380.594,Z 745.328,A -85,B 0,C 180,E1 -12177.832,E2 -12177.832} C_VEL
LIN {X 0,Y 379.901,Z 755.801,A -85,B 0,C 180,E1 -12178.605,E2 -12178.605} C_VEL
LIN {X 0,Y 379.001,Z 767.538,A -85,B 0,C 180,E1 -12179.705,E2 -12179.705} C_VEL
LIN {X 0,Y 378.091,Z 778.151,A -85,B 0,C 180,E1 -12180.964,E2 -12180.964} C_VEL
LIN {X 0,Y 377.271,Z 787.727,A -85,B 0,C 180,E1 -12182.382,E2 -12182.382} C_VEL
LIN {X 0,Y 376.529,Z 795.397,A -85,B 0,C 180,E1 -12183.769,E2 -12183.769} C_VEL
LIN {X 0,Y 375.857,Z 802.83,A -85,B 0,C 180,E1 -12185.425,E2 -12185.425} C_VEL
LIN {X 0,Y 375.385,Z 808.811,A -85,B 0,C 180,E1 -12187.122,E2 -12187.122} C_VEL
LIN {X 0,Y 374.985,Z 813.631,A -85,B 0,C 180,E1 -12188.891,E2 -12188.891} C_VEL
LIN {X 0,Y 374.718,Z 816.655,A -85,B 0,C 180,E1 -12190.358,E2 -12190.358} C_VEL
LIN {X 0,Y 374.512,Z 819.593,A -85,B 0,C 180,E1 -12192.497,E2 -12192.497} C_VEL
LIN {X 0,Y 374.383,Z 820.864,A -85,B 0,C 180,E1 -12194.493,E2 -12194.493} C_VEL
LIN {X 0,Y 374.402,Z 820.904,A -85,B 0,C 180,E1 -12196.011,E2 -12196.011} C_VEL
LIN {X 0,Y 374.52,Z 820.136,A -85,B 0,C 180,E1 -12197.504,E2 -12197.504} C_VEL
LIN {X 0,Y 374.643,Z 818.653,A -85,B 0,C 180,E1 -12198.962,E2 -12198.962} C_VEL
LIN {X 0,Y 374.908,Z 816.441,A -85,B 0,C 180,E1 -12200.405,E2 -12200.405} C_VEL
LIN {X 0,Y 375.22,Z 813.348,A -85,B 0,C 180,E1 -12201.874,E2 -12201.874} C_VEL
LIN {X 0,Y 375.666,Z 808.711,A -85,B 0,C 180,E1 -12203.555,E2 -12203.555} C_VEL
LIN {X 0,Y 376.298,Z 802.612,A -85,B 0,C 180,E1 -12205.261,E2 -12205.261} C_VEL
LIN {X 0,Y 377.099,Z 794.74,A -85,B 0,C 180,E1 -12206.997,E2 -12206.997} C_VEL
LIN {X 0,Y 378.051,Z 786.345,A -85,B 0,C 180,E1 -12208.477,E2 -12208.477} C_VEL
LIN {X 0,Y 378.974,Z 777.071,A -85,B 0,C 180,E1 -12209.8,E2 -12209.8} C_VEL
LIN {X 0,Y 379.924,Z 766.676,A -85,B 0,C 180,E1 -12211,E2 -12211} C_VEL
LIN {X 0,Y 380.854,Z 756.064,A -85,B 0,C 180,E1 -12211.981,E2 -12211.981} C_VEL
LIN {X 0,Y 381.65,Z 744.691,A -85,B 0,C 180,E1 -12212.812,E2 -12212.812} C_VEL
LIN {X 0,Y 382.34,Z 731.708,A -85,B 0,C 180,E1 -12213.511,E2 -12213.511} C_VEL
LIN {X 0,Y 382.791,Z 718.644,A -85,B 0,C 180,E1 -12213.99,E2 -12213.99} C_VEL
LIN {X 0,Y 384.533,Z 633.612,A -85,B 0,C 180,E1 -12215.748,E2 -12215.748} C_VEL
LIN {X 0,Y 381.864,Z 622.484,A -85,B 0,C 180,E1 -12216.17,E2 -12216.17} C_VEL
LIN {X 0,Y 377.77,Z 612.202,A -85,B 0,C 180,E1 -12216.714,E2 -12216.714} C_VEL
LIN {X 0,Y 376.024,Z 603.646,A -85,B 0,C 180,E1 -12219.436,E2 -12219.436} C_VEL
LIN {X 0,Y 376.041,Z 603.646,A -85,B 0,C 180,E1 -12222.601,E2 -12222.601} C_VEL
LIN {X 0,Y 376.081,Z 603.64,A -85,B 0,C 180,E1 -12226.342,E2 -12226.342} C_VEL
LIN {X 0,Y 376.115,Z 603.637,A -85,B 0,C 180,E1 -12230.319,E2 -12230.319} C_VEL
LIN {X 0,Y 376.222,Z 603.622,A -85,B 0,C 180,E1 -12232.487,E2 -12232.487} C_VEL
LIN {X 0,Y 376.171,Z 603.628,A -85,B 0,C 180,E1 -12234.64,E2 -12234.64} C_VEL
LIN {X 0,Y 376.35,Z 603.604,A -85,B 0,C 180,E1 -12237.86,E2 -12237.86} C_VEL
LIN {X 0,Y 376.482,Z 603.587,A -85,B 0,C 180,E1 -12240.001,E2 -12240.001} C_VEL
LIN {X 0,Y 376.184,Z 603.623,A -85,B 0,C 180,E1 -12243.213,E2 -12243.213} C_VEL
LIN {X 0,Y 376.246,Z 603.617,A -85,B 0,C 180,E1 -12246.436,E2 -12246.436} C_VEL
LIN {X 0,Y 376.198,Z 603.625,A -85,B 0,C 180,E1 -12248.596,E2 -12248.596} C_VEL
LIN {X 0,Y 376.052,Z 603.639,A -85,B 0,C 180,E1 -12251.864,E2 -12251.864} C_VEL
LIN {X 0,Y 376.052,Z 603.64,A -85,B 0,C 180,E1 -12255.168,E2 -12255.168} C_VEL
LIN {X 0,Y 376.002,Z 603.647,A -85,B 0,C 180,E1 -12258.528,E2 -12258.528} C_VEL
LIN {X 0,Y 375.956,Z 603.649,A -85,B 0,C 180,E1 -12261.955,E2 -12261.955} C_VEL
LIN {X 0,Y 376,Z 603.643,A -85,B 0,C 180,E1 -12265.462,E2 -12265.462} C_VEL
LIN {X 0,Y 375.972,Z 603.647,A -85,B 0,C 180,E1 -12269.08,E2 -12269.08} C_VEL
LIN {X 0,Y 375.952,Z 603.648,A -85,B 0,C 180,E1 -12272.829,E2 -12272.829} C_VEL
LIN {X 0,Y 375.954,Z 603.65,A -85,B 0,C 180,E1 -12275.416,E2 -12275.416} C_VEL
LIN {X 0,Y 375.973,Z 603.647,A -85,B 0,C 180,E1 -12278.272,E2 -12278.272} C_VEL
LIN {X 0,Y 375.957,Z 603.654,A -85,B 0,C 180,E1 -12281.606,E2 -12281.606} C_VEL
LIN {X 0,Y 375.951,Z 603.657,A -85,B 0,C 180,E1 -12285.266,E2 -12285.266} C_VEL
LIN {X 0,Y 375.979,Z 603.653,A -85,B 0,C 180,E1 -12289.139,E2 -12289.139} C_VEL
LIN {X 0,Y 375.967,Z 603.654,A -85,B 0,C 180,E1 -12291.913,E2 -12291.913} C_VEL
LIN {X 0,Y 375.98,Z 603.655,A -85,B 0,C 180,E1 -12295.334,E2 -12295.334} C_VEL
LIN {X 0,Y 375.982,Z 603.821,A -85,B 0,C 180,E1 -12299.113,E2 -12299.113} C_VEL
LIN {X 0,Y 378.615,Z 615.104,A -85,B 0,C 180,E1 -12302.051,E2 -12302.051} C_VEL
LIN {X 0,Y 380.292,Z 624.164,A -85,B 0,C 180,E1 -12304.26,E2 -12304.26} C_VEL
LIN {X 0,Y 379.602,Z 631.91,A -85,B 0,C 180,E1 -12305.965,E2 -12305.965} C_VEL
LIN {X 0,Y 378.567,Z 643.182,A -85,B 0,C 180,E1 -12308.39,E2 -12308.39} C_VEL
LIN {X 0,Y 382.006,Z 663.273,A -85,B 0,C 180,E1 -12309.062,E2 -12309.062} C_VEL
LIN {X 0,Y 383.921,Z 678.183,A -85,B 0,C 180,E1 -12309.507,E2 -12309.507} C_VEL
LIN {X 0,Y 382.523,Z 752.28,A -85,B 0,C 180,E1 -12311.037,E2 -12311.037} C_VEL
LIN {X 0,Y 381.771,Z 765.971,A -85,B 0,C 180,E1 -12311.52,E2 -12311.52} C_VEL
LIN {X 0,Y 380.87,Z 778.97,A -85,B 0,C 180,E1 -12312.205,E2 -12312.205} C_VEL
LIN {X 0,Y 379.937,Z 790.823,A -85,B 0,C 180,E1 -12313.062,E2 -12313.062} C_VEL
LIN {X 0,Y 378.833,Z 802.282,A -85,B 0,C 180,E1 -12314.12,E2 -12314.12} C_VEL
LIN {X 0,Y 377.938,Z 811.967,A -85,B 0,C 180,E1 -12315.235,E2 -12315.235} C_VEL
LIN {X 0,Y 377.068,Z 821.161,A -85,B 0,C 180,E1 -12316.528,E2 -12316.528} C_VEL
LIN {X 0,Y 376.133,Z 830.406,A -85,B 0,C 180,E1 -12318.14,E2 -12318.14} C_VEL
LIN {X 0,Y 375.442,Z 837.879,A -85,B 0,C 180,E1 -12319.757,E2 -12319.757} C_VEL
LIN {X 0,Y 375.003,Z 843.888,A -85,B 0,C 180,E1 -12321.377,E2 -12321.377} C_VEL
LIN {X 0,Y 374.733,Z 848.635,A -85,B 0,C 180,E1 -12322.998,E2 -12322.998} C_VEL
LIN {X 0,Y 374.577,Z 852.259,A -85,B 0,C 180,E1 -12324.617,E2 -12324.617} C_VEL
LIN {X 0,Y 374.577,Z 854.098,A -85,B 0,C 180,E1 -12325.696,E2 -12325.696} C_VEL
LIN {X 0,Y 374.575,Z 856.5,A -85,B 0,C 180,E1 -12327.85,E2 -12327.85} C_VEL
LIN {X 0,Y 374.624,Z 857.098,A -85,B 0,C 180,E1 -12328.925,E2 -12328.925} C_VEL
LIN {X 0,Y 374.608,Z 857.245,A -85,B 0,C 180,E1 -12330,E2 -12330} C_VEL
LIN {X 0,Y 374.625,Z 856.987,A -85,B 0,C 180,E1 -12331.075,E2 -12331.075} C_VEL
LIN {X 0,Y 374.589,Z 856.329,A -85,B 0,C 180,E1 -12332.15,E2 -12332.15} C_VEL
LIN {X 0,Y 374.51,Z 855.26,A -85,B 0,C 180,E1 -12333.227,E2 -12333.227} C_VEL
LIN {X 0,Y 374.571,Z 853.729,A -85,B 0,C 180,E1 -12334.304,E2 -12334.304} C_VEL
LIN {X 0,Y 374.595,Z 850.242,A -85,B 0,C 180,E1 -12336.082,E2 -12336.082} C_VEL
LIN {X 0,Y 374.87,Z 844.773,A -85,B 0,C 180,E1 -12338.083,E2 -12338.083} C_VEL
LIN {X 0,Y 375.325,Z 837.804,A -85,B 0,C 180,E1 -12339.974,E2 -12339.974} C_VEL
LIN {X 0,Y 375.94,Z 830.238,A -85,B 0,C 180,E1 -12341.593,E2 -12341.593} C_VEL
LIN {X 0,Y 376.639,Z 822.515,A -85,B 0,C 180,E1 -12342.939,E2 -12342.939} C_VEL
LIN {X 0,Y 377.423,Z 812.958,A -85,B 0,C 180,E1 -12344.304,E2 -12344.304} C_VEL
LIN {X 0,Y 378.394,Z 801.366,A -85,B 0,C 180,E1 -12345.623,E2 -12345.623} C_VEL
LIN {X 0,Y 379.441,Z 789.437,A -85,B 0,C 180,E1 -12346.683,E2 -12346.683} C_VEL
LIN {X 0,Y 380.218,Z 777.804,A -85,B 0,C 180,E1 -12347.479,E2 -12347.479} C_VEL
LIN {X 0,Y 381.085,Z 764.75,A -85,B 0,C 180,E1 -12348.132,E2 -12348.132} C_VEL
LIN {X 0,Y 381.619,Z 751.91,A -85,B 0,C 180,E1 -12348.557,E2 -12348.557} C_VEL
LIN {X 0,Y 382.793,Z 676.636,A -85,B 0,C 180,E1 -12350.074,E2 -12350.074} C_VEL
LIN {X 0,Y 378.141,Z 644.639,A -85,B 0,C 180,E1 -12350.999,E2 -12350.999} C_VEL
LIN {X 0,Y 379.855,Z 625.915,A -85,B 0,C 180,E1 -12354.961,E2 -12354.961} C_VEL
LIN {X 0,Y 379.815,Z 622.219,A -85,B 0,C 180,E1 -12355.774,E2 -12355.774} C_VEL
LIN {X 0,Y 377.656,Z 611.314,A -85,B 0,C 180,E1 -12358.329,E2 -12358.329} C_VEL
LIN {X 0,Y 375.986,Z 603.652,A -85,B 0,C 180,E1 -12360.232,E2 -12360.232} C_VEL
LIN {X 0,Y 375.96,Z 603.653,A -85,B 0,C 180,E1 -12364.11,E2 -12364.11} C_VEL
LIN {X 0,Y 375.955,Z 603.654,A -85,B 0,C 180,E1 -12366.74,E2 -12366.74} C_VEL
LIN {X 0,Y 375.996,Z 603.646,A -85,B 0,C 180,E1 -12369.971,E2 -12369.971} C_VEL
LIN {X 0,Y 375.936,Z 603.653,A -85,B 0,C 180,E1 -12373.764,E2 -12373.764} C_VEL
LIN {X 0,Y 375.958,Z 603.65,A -85,B 0,C 180,E1 -12377.703,E2 -12377.703} C_VEL
LIN {X 0,Y 375.965,Z 603.654,A -85,B 0,C 180,E1 -12380.537,E2 -12380.537} C_VEL
LIN {X 0,Y 375.963,Z 603.65,A -85,B 0,C 180,E1 -12383.494,E2 -12383.494} C_VEL
LIN {X 0,Y 375.956,Z 603.65,A -85,B 0,C 180,E1 -12385.888,E2 -12385.888} C_VEL
LIN {X 0,Y 375.965,Z 603.649,A -85,B 0,C 180,E1 -12389.687,E2 -12389.687} C_VEL
LIN {X 0,Y 375.997,Z 603.645,A -85,B 0,C 180,E1 -12392.141,E2 -12392.141} C_VEL
LIN {X 0,Y 375.999,Z 603.647,A -85,B 0,C 180,E1 -12394.538,E2 -12394.538} C_VEL
LIN {X 0,Y 375.951,Z 603.651,A -85,B 0,C 180,E1 -12398.044,E2 -12398.044} C_VEL
LIN {X 0,Y 376.002,Z 603.648,A -85,B 0,C 180,E1 -12401.472,E2 -12401.472} C_VEL
LIN {X 0,Y 376.05,Z 603.641,A -85,B 0,C 180,E1 -12404.832,E2 -12404.832} C_VEL
LIN {X 0,Y 376.042,Z 603.639,A -85,B 0,C 180,E1 -12408.136,E2 -12408.136} C_VEL
LIN {X 0,Y 376.211,Z 603.619,A -85,B 0,C 180,E1 -12411.918,E2 -12411.918} C_VEL
LIN {X 0,Y 376.165,Z 603.625,A -85,B 0,C 180,E1 -12414.639,E2 -12414.639} C_VEL
LIN {X 0,Y 376.345,Z 603.604,A -85,B 0,C 180,E1 -12417.859,E2 -12417.859} C_VEL
LIN {X 0,Y 376.482,Z 603.586,A -85,B 0,C 180,E1 -12419.999,E2 -12419.999} C_VEL
LIN {X 0,Y 376.184,Z 603.625,A -85,B 0,C 180,E1 -12423.212,E2 -12423.212} C_VEL
LIN {X 0,Y 376.224,Z 603.617,A -85,B 0,C 180,E1 -12426.605,E2 -12426.605} C_VEL
LIN {X 0,Y 376.113,Z 603.637,A -85,B 0,C 180,E1 -12429.681,E2 -12429.681} C_VEL
LIN {X 0,Y 376.08,Z 603.641,A -85,B 0,C 180,E1 -12433.657,E2 -12433.657} C_VEL
LIN {X 0,Y 376.034,Z 603.646,A -85,B 0,C 180,E1 -12437.607,E2 -12437.607} C_VEL
LIN {X 0,Y 375.969,Z 603.648,A -85,B 0,C 180,E1 -12440.832,E2 -12440.832} C_VEL
LIN {X 0,Y 375.984,Z 603.649,A -85,B 0,C 180,E1 -12444.281,E2 -12444.281} C_VEL
LIN {X 0,Y 376.011,Z 603.644,A -85,B 0,C 180,E1 -12446.652,E2 -12446.652} C_VEL
LIN {X 0,Y 375.968,Z 603.649,A -85,B 0,C 180,E1 -12449.079,E2 -12449.079} C_VEL
LIN {X 0,Y 375.949,Z 603.651,A -85,B 0,C 180,E1 -12452.828,E2 -12452.828} C_VEL
LIN {X 0,Y 375.95,Z 603.652,A -85,B 0,C 180,E1 -12455.416,E2 -12455.416} C_VEL
LIN {X 0,Y 375.97,Z 603.654,A -85,B 0,C 180,E1 -12458.272,E2 -12458.272} C_VEL
LIN {X 0,Y 375.982,Z 603.648,A -85,B 0,C 180,E1 -12461.611,E2 -12461.611} C_VEL
LIN {X 0,Y 375.964,Z 603.649,A -85,B 0,C 180,E1 -12465.262,E2 -12465.262} C_VEL
LIN {X 0,Y 375.971,Z 603.648,A -85,B 0,C 180,E1 -12469.138,E2 -12469.138} C_VEL
LIN {X 0,Y 375.96,Z 603.652,A -85,B 0,C 180,E1 -12471.912,E2 -12471.912} C_VEL
LIN {X 0,Y 375.974,Z 603.648,A -85,B 0,C 180,E1 -12475.333,E2 -12475.333} C_VEL
LIN {X 0,Y 375.952,Z 603.657,A -85,B 0,C 180,E1 -12478.438,E2 -12478.438} C_VEL
LIN {X 0,Y 375.978,Z 603.65,A -85,B 0,C 180,E1 -12482.141,E2 -12482.141} C_VEL
LIN {X 0,Y 376.002,Z 603.651,A -85,B 0,C 180,E1 -12484.539,E2 -12484.539} C_VEL
LIN {X 0,Y 375.963,Z 603.65,A -85,B 0,C 180,E1 -12488.046,E2 -12488.046} C_VEL
LIN {X 0,Y 376.005,Z 603.645,A -85,B 0,C 180,E1 -12491.474,E2 -12491.474} C_VEL
LIN {X 0,Y 376.056,Z 603.645,A -85,B 0,C 180,E1 -12494.833,E2 -12494.833} C_VEL
LIN {X 0,Y 376.047,Z 603.639,A -85,B 0,C 180,E1 -12498.137,E2 -12498.137} C_VEL
LIN {X 0,Y 376.215,Z 603.618,A -85,B 0,C 180,E1 -12501.919,E2 -12501.919} C_VEL
LIN {X 0,Y 376.167,Z 603.627,A -85,B 0,C 180,E1 -12504.64,E2 -12504.64} C_VEL
LIN {X 0,Y 376.351,Z 603.601,A -85,B 0,C 180,E1 -12507.86,E2 -12507.86} C_VEL
LIN {X 0,Y 376.486,Z 603.584,A -85,B 0,C 180,E1 -12510,E2 -12510} C_VEL
LIN {X 0,Y 376.187,Z 603.628,A -85,B 0,C 180,E1 -12513.213,E2 -12513.213} C_VEL
LIN {X 0,Y 376.235,Z 603.616,A -85,B 0,C 180,E1 -12516.435,E2 -12516.435} C_VEL
LIN {X 0,Y 376.116,Z 603.633,A -85,B 0,C 180,E1 -12519.681,E2 -12519.681} C_VEL
LIN {X 0,Y 376.085,Z 603.637,A -85,B 0,C 180,E1 -12523.657,E2 -12523.657} C_VEL
LIN {X 0,Y 376.039,Z 603.646,A -85,B 0,C 180,E1 -12527.607,E2 -12527.607} C_VEL
LIN {X 0,Y 375.972,Z 603.654,A -85,B 0,C 180,E1 -12530.831,E2 -12530.831} C_VEL
LIN {X 0,Y 376.009,Z 603.691,A -85,B 0,C 180,E1 -12532.095,E2 -12532.095} C_VEL
LIN {X 0,Y 377.347,Z 610.438,A -85,B 0,C 180,E1 -12534.046,E2 -12534.046} C_VEL
LIN {X 0,Y 380.901,Z 621.68,A -85,B 0,C 180,E1 -12534.492,E2 -12534.492} C_VEL
LIN {X 0,Y 383.35,Z 633.495,A -85,B 0,C 180,E1 -12534.866,E2 -12534.866} C_VEL
LIN {X 0,Y 382.084,Z 699.975,A -85,B 0,C 180,E1 -12536.184,E2 -12536.184} C_VEL
LIN {X 0,Y 381.319,Z 703.897,A -85,B 0,C 180,E1 -12536.229,E2 -12536.229} C_VEL
LIN {X 0,Y 375.505,Z 716.126,A -85,B 0,C 180,E1 -12536.235,E2 -12536.235} C_VEL
LIN {X 0,Y 374.879,Z 719.998,A -85,B 0,C 180,E1 -12536.323,E2 -12536.323} C_VEL
LIN {X 0,Y 374.451,Z 733.303,A -85,B 0,C 180,E1 -12536.847,E2 -12536.847} C_VEL
LIN {X 0,Y 373.783,Z 745.119,A -85,B 0,C 180,E1 -12537.519,E2 -12537.519} C_VEL
LIN {X 0,Y 372.973,Z 756.93,A -85,B 0,C 180,E1 -12538.41,E2 -12538.41} C_VEL
LIN {X 0,Y 372.016,Z 768.721,A -85,B 0,C 180,E1 -12539.551,E2 -12539.551} C_VEL
LIN {X 0,Y 371.147,Z 778.518,A -85,B 0,C 180,E1 -12540.748,E2 -12540.748} C_VEL
LIN {X 0,Y 370.248,Z 788.543,A -85,B 0,C 180,E1 -12542.266,E2 -12542.266} C_VEL
LIN {X 0,Y 369.416,Z 796.79,A -85,B 0,C 180,E1 -12543.811,E2 -12543.811} C_VEL
LIN {X 0,Y 368.725,Z 804.268,A -85,B 0,C 180,E1 -12545.58,E2 -12545.58} C_VEL
LIN {X 0,Y 368.293,Z 809.586,A -85,B 0,C 180,E1 -12547.16,E2 -12547.16} C_VEL
LIN {X 0,Y 367.855,Z 814.593,A -85,B 0,C 180,E1 -12549.084,E2 -12549.084} C_VEL
LIN {X 0,Y 367.619,Z 817.381,A -85,B 0,C 180,E1 -12550.54,E2 -12550.54} C_VEL
LIN {X 0,Y 367.47,Z 819.44,A -85,B 0,C 180,E1 -12552.019,E2 -12552.019} C_VEL
LIN {X 0,Y 367.351,Z 820.775,A -85,B 0,C 180,E1 -12553.529,E2 -12553.529} C_VEL
LIN {X 0,Y 367.295,Z 821.31,A -85,B 0,C 180,E1 -12555.069,E2 -12555.069} C_VEL
LIN {X 0,Y 367.367,Z 821.045,A -85,B 0,C 180,E1 -12556.631,E2 -12556.631} C_VEL
LIN {X 0,Y 367.493,Z 819.938,A -85,B 0,C 180,E1 -12558.23,E2 -12558.23} C_VEL
LIN {X 0,Y 367.697,Z 817.906,A -85,B 0,C 180,E1 -12559.865,E2 -12559.865} C_VEL
LIN {X 0,Y 368.059,Z 814.854,A -85,B 0,C 180,E1 -12561.524,E2 -12561.524} C_VEL
LIN {X 0,Y 368.495,Z 810.6,A -85,B 0,C 180,E1 -12563.227,E2 -12563.227} C_VEL
LIN {X 0,Y 369.23,Z 804.162,A -85,B 0,C 180,E1 -12565.179,E2 -12565.179} C_VEL
LIN {X 0,Y 369.91,Z 797.728,A -85,B 0,C 180,E1 -12566.714,E2 -12566.714} C_VEL
LIN {X 0,Y 370.849,Z 789.725,A -85,B 0,C 180,E1 -12568.255,E2 -12568.255} C_VEL
LIN {X 0,Y 371.782,Z 781.408,A -85,B 0,C 180,E1 -12569.565,E2 -12569.565} C_VEL
LIN {X 0,Y 372.879,Z 770.426,A -85,B 0,C 180,E1 -12570.966,E2 -12570.966} C_VEL
LIN {X 0,Y 373.894,Z 759.603,A -85,B 0,C 180,E1 -12572.059,E2 -12572.059} C_VEL
LIN {X 0,Y 374.864,Z 747.146,A -85,B 0,C 180,E1 -12573.034,E2 -12573.034} C_VEL
LIN {X 0,Y 375.624,Z 734.583,A -85,B 0,C 180,E1 -12573.771,E2 -12573.771} C_VEL
LIN {X 0,Y 376.084,Z 722.923,A -85,B 0,C 180,E1 -12574.253,E2 -12574.253} C_VEL
LIN {X 0,Y 376.519,Z 706.75,A -85,B 0,C 180,E1 -12574.651,E2 -12574.651} C_VEL
LIN {X 0,Y 378.024,Z 634.883,A -85,B 0,C 180,E1 -12576.15,E2 -12576.15} C_VEL
LIN {X 0,Y 375.659,Z 624.965,A -85,B 0,C 180,E1 -12576.539,E2 -12576.539} C_VEL
LIN {X 0,Y 370.655,Z 612.682,A -85,B 0,C 180,E1 -12577.201,E2 -12577.201} C_VEL
LIN {X 0,Y 368.968,Z 604.525,A -85,B 0,C 180,E1 -12579.815,E2 -12579.815} C_VEL
LIN {X 0,Y 368.966,Z 604.524,A -85,B 0,C 180,E1 -12583.399,E2 -12583.399} C_VEL
LIN {X 0,Y 369.051,Z 604.517,A -85,B 0,C 180,E1 -12586.791,E2 -12586.791} C_VEL
LIN {X 0,Y 369.064,Z 604.515,A -85,B 0,C 180,E1 -12590.132,E2 -12590.132} C_VEL
LIN {X 0,Y 369.18,Z 604.499,A -85,B 0,C 180,E1 -12592.343,E2 -12592.343} C_VEL
LIN {X 0,Y 369.143,Z 604.503,A -85,B 0,C 180,E1 -12594.538,E2 -12594.538} C_VEL
LIN {X 0,Y 369.316,Z 604.48,A -85,B 0,C 180,E1 -12597.819,E2 -12597.819} C_VEL
LIN {X 0,Y 369.451,Z 604.463,A -85,B 0,C 180,E1 -12600.001,E2 -12600.001} C_VEL
LIN {X 0,Y 369.311,Z 604.48,A -85,B 0,C 180,E1 -12602.182,E2 -12602.182} C_VEL
LIN {X 0,Y 369.206,Z 604.493,A -85,B 0,C 180,E1 -12606.559,E2 -12606.559} C_VEL
LIN {X 0,Y 369.132,Z 604.506,A -85,B 0,C 180,E1 -12608.762,E2 -12608.762} C_VEL
LIN {X 0,Y 369.006,Z 604.517,A -85,B 0,C 180,E1 -12612.094,E2 -12612.094} C_VEL
LIN {X 0,Y 368.991,Z 604.517,A -85,B 0,C 180,E1 -12615.466,E2 -12615.466} C_VEL
LIN {X 0,Y 368.951,Z 604.525,A -85,B 0,C 180,E1 -12618.895,E2 -12618.895} C_VEL
LIN {X 0,Y 368.925,Z 604.525,A -85,B 0,C 180,E1 -12622.396,E2 -12622.396} C_VEL
LIN {X 0,Y 368.994,Z 604.515,A -85,B 0,C 180,E1 -12625.981,E2 -12625.981} C_VEL
LIN {X 0,Y 368.962,Z 604.52,A -85,B 0,C 180,E1 -12628.814,E2 -12628.814} C_VEL
LIN {X 0,Y 368.905,Z 604.524,A -85,B 0,C 180,E1 -12632.238,E2 -12632.238} C_VEL
LIN {X 0,Y 368.925,Z 604.525,A -85,B 0,C 180,E1 -12635.003,E2 -12635.003} C_VEL
LIN {X 0,Y 368.908,Z 604.527,A -85,B 0,C 180,E1 -12638.642,E2 -12638.642} C_VEL
LIN {X 0,Y 368.907,Z 604.534,A -85,B 0,C 180,E1 -12641.82,E2 -12641.82} C_VEL
LIN {X 0,Y 368.924,Z 604.533,A -85,B 0,C 180,E1 -12645.184,E2 -12645.184} C_VEL
LIN {X 0,Y 368.908,Z 604.531,A -85,B 0,C 180,E1 -12648.182,E2 -12648.182} C_VEL
LIN {X 0,Y 368.912,Z 604.533,A -85,B 0,C 180,E1 -12651.36,E2 -12651.36} C_VEL
LIN {X 0,Y 368.937,Z 604.531,A -85,B 0,C 180,E1 -12655.148,E2 -12655.148} C_VEL
LIN {X 0,Y 368.939,Z 604.651,A -85,B 0,C 180,E1 -12658.65,E2 -12658.65} C_VEL
LIN {X 0,Y 371.697,Z 616.404,A -85,B 0,C 180,E1 -12661.791,E2 -12661.791} C_VEL
LIN {X 0,Y 373.355,Z 625.38,A -85,B 0,C 180,E1 -12664.046,E2 -12664.046} C_VEL
LIN {X 0,Y 373.136,Z 629.885,A -85,B 0,C 180,E1 -12665.072,E2 -12665.072} C_VEL
LIN {X 0,Y 371.771,Z 642.743,A -85,B 0,C 180,E1 -12667.908,E2 -12667.908} C_VEL
LIN {X 0,Y 375.326,Z 663.038,A -85,B 0,C 180,E1 -12668.623,E2 -12668.623} C_VEL
LIN {X 0,Y 377.362,Z 678.319,A -85,B 0,C 180,E1 -12669.099,E2 -12669.099} C_VEL
LIN {X 0,Y 375.877,Z 752.099,A -85,B 0,C 180,E1 -12670.653,E2 -12670.653} C_VEL
LIN {X 0,Y 375.113,Z 765.698,A -85,B 0,C 180,E1 -12671.145,E2 -12671.145} C_VEL
LIN {X 0,Y 374.203,Z 778.1,A -85,B 0,C 180,E1 -12671.806,E2 -12671.806} C_VEL
LIN {X 0,Y 373.307,Z 789.262,A -85,B 0,C 180,E1 -12672.611,E2 -12672.611} C_VEL
LIN {X 0,Y 372.124,Z 800.912,A -85,B 0,C 180,E1 -12673.685,E2 -12673.685} C_VEL
LIN {X 0,Y 371.132,Z 810.959,A -85,B 0,C 180,E1 -12674.845,E2 -12674.845} C_VEL
LIN {X 0,Y 370.119,Z 820.976,A -85,B 0,C 180,E1 -12676.27,E2 -12676.27} C_VEL
LIN {X 0,Y 369.151,Z 830.195,A -85,B 0,C 180,E1 -12677.912,E2 -12677.912} C_VEL
LIN {X 0,Y 368.42,Z 837.647,A -85,B 0,C 180,E1 -12679.559,E2 -12679.559} C_VEL
LIN {X 0,Y 367.938,Z 843.635,A -85,B 0,C 180,E1 -12681.211,E2 -12681.211} C_VEL
LIN {X 0,Y 367.662,Z 848.362,A -85,B 0,C 180,E1 -12682.863,E2 -12682.863} C_VEL
LIN {X 0,Y 367.488,Z 851.97,A -85,B 0,C 180,E1 -12684.513,E2 -12684.513} C_VEL
LIN {X 0,Y 367.481,Z 853.791,A -85,B 0,C 180,E1 -12685.613,E2 -12685.613} C_VEL
LIN {X 0,Y 367.475,Z 856.175,A -85,B 0,C 180,E1 -12687.808,E2 -12687.808} C_VEL
LIN {X 0,Y 367.54,Z 856.76,A -85,B 0,C 180,E1 -12688.904,E2 -12688.904} C_VEL
LIN {X 0,Y 367.541,Z 856.894,A -85,B 0,C 180,E1 -12690,E2 -12690} C_VEL
LIN {X 0,Y 367.559,Z 856.628,A -85,B 0,C 180,E1 -12691.096,E2 -12691.096} C_VEL
LIN {X 0,Y 367.49,Z 855.959,A -85,B 0,C 180,E1 -12692.192,E2 -12692.192} C_VEL
LIN {X 0,Y 367.425,Z 854.874,A -85,B 0,C 180,E1 -12693.29,E2 -12693.29} C_VEL
LIN {X 0,Y 367.498,Z 853.329,A -85,B 0,C 180,E1 -12694.387,E2 -12694.387} C_VEL
LIN {X 0,Y 367.497,Z 850.189,A -85,B 0,C 180,E1 -12696.037,E2 -12696.037} C_VEL
LIN {X 0,Y 367.702,Z 845.961,A -85,B 0,C 180,E1 -12697.689,E2 -12697.689} C_VEL
LIN {X 0,Y 368.132,Z 839.5,A -85,B 0,C 180,E1 -12699.616,E2 -12699.616} C_VEL
LIN {X 0,Y 368.69,Z 832.436,A -85,B 0,C 180,E1 -12701.267,E2 -12701.267} C_VEL
LIN {X 0,Y 369.532,Z 823.571,A -85,B 0,C 180,E1 -12702.913,E2 -12702.913} C_VEL
LIN {X 0,Y 370.411,Z 813.268,A -85,B 0,C 180,E1 -12704.45,E2 -12704.45} C_VEL
LIN {X 0,Y 371.388,Z 801.896,A -85,B 0,C 180,E1 -12705.785,E2 -12705.785} C_VEL
LIN {X 0,Y 372.461,Z 790.223,A -85,B 0,C 180,E1 -12706.864,E2 -12706.864} C_VEL
LIN {X 0,Y 373.346,Z 777.826,A -85,B 0,C 180,E1 -12707.741,E2 -12707.741} C_VEL
LIN {X 0,Y 374.234,Z 764.894,A -85,B 0,C 180,E1 -12708.405,E2 -12708.405} C_VEL
LIN {X 0,Y 374.771,Z 752.448,A -85,B 0,C 180,E1 -12708.838,E2 -12708.838} C_VEL
LIN {X 0,Y 376.03,Z 677.552,A -85,B 0,C 180,E1 -12710.38,E2 -12710.38} C_VEL
LIN {X 0,Y 371.24,Z 644.387,A -85,B 0,C 180,E1 -12711.357,E2 -12711.357} C_VEL
LIN {X 0,Y 372.99,Z 626.308,A -85,B 0,C 180,E1 -12715.252,E2 -12715.252} C_VEL
LIN {X 0,Y 372.55,Z 621.665,A -85,B 0,C 180,E1 -12716.315,E2 -12716.315} C_VEL
LIN {X 0,Y 370.127,Z 609.981,A -85,B 0,C 180,E1 -12719.137,E2 -12719.137} C_VEL
LIN {X 0,Y 368.923,Z 604.532,A -85,B 0,C 180,E1 -12720.517,E2 -12720.517} C_VEL
LIN {X 0,Y 368.896,Z 604.531,A -85,B 0,C 180,E1 -12723.537,E2 -12723.537} C_VEL
LIN {X 0,Y 368.903,Z 604.532,A -85,B 0,C 180,E1 -12726.855,E2 -12726.855} C_VEL
LIN {X 0,Y 368.952,Z 604.527,A -85,B 0,C 180,E1 -12730.364,E2 -12730.364} C_VEL
LIN {X 0,Y 368.892,Z 604.53,A -85,B 0,C 180,E1 -12733.617,E2 -12733.617} C_VEL
LIN {X 0,Y 368.902,Z 604.536,A -85,B 0,C 180,E1 -12736.698,E2 -12736.698} C_VEL
LIN {X 0,Y 368.95,Z 604.523,A -85,B 0,C 180,E1 -12739.634,E2 -12739.634} C_VEL
LIN {X 0,Y 368.903,Z 604.532,A -85,B 0,C 180,E1 -12743.142,E2 -12743.142} C_VEL
LIN {X 0,Y 368.895,Z 604.532,A -85,B 0,C 180,E1 -12746.461,E2 -12746.461} C_VEL
LIN {X 0,Y 368.919,Z 604.528,A -85,B 0,C 180,E1 -12750.309,E2 -12750.309} C_VEL
LIN {X 0,Y 368.976,Z 604.521,A -85,B 0,C 180,E1 -12753.534,E2 -12753.534} C_VEL
LIN {X 0,Y 368.95,Z 604.524,A -85,B 0,C 180,E1 -12756.42,E2 -12756.42} C_VEL
LIN {X 0,Y 368.929,Z 604.526,A -85,B 0,C 180,E1 -12759.946,E2 -12759.946} C_VEL
LIN {X 0,Y 368.968,Z 604.525,A -85,B 0,C 180,E1 -12763.398,E2 -12763.398} C_VEL
LIN {X 0,Y 369.05,Z 604.513,A -85,B 0,C 180,E1 -12766.789,E2 -12766.789} C_VEL
LIN {X 0,Y 369.06,Z 604.509,A -85,B 0,C 180,E1 -12770.131,E2 -12770.131} C_VEL
LIN {X 0,Y 369.155,Z 604.497,A -85,B 0,C 180,E1 -12772.341,E2 -12772.341} C_VEL
LIN {X 0,Y 369.137,Z 604.5,A -85,B 0,C 180,E1 -12774.537,E2 -12774.537} C_VEL
LIN {X 0,Y 369.31,Z 604.481,A -85,B 0,C 180,E1 -12777.818,E2 -12777.818} C_VEL
LIN {X 0,Y 369.451,Z 604.462,A -85,B 0,C 180,E1 -12779.999,E2 -12779.999} C_VEL
LIN {X 0,Y 369.311,Z 604.479,A -85,B 0,C 180,E1 -12782.181,E2 -12782.181} C_VEL
LIN {X 0,Y 369.195,Z 604.492,A -85,B 0,C 180,E1 -12786.589,E2 -12786.589} C_VEL
LIN {X 0,Y 369.061,Z 604.513,A -85,B 0,C 180,E1 -12789.868,E2 -12789.868} C_VEL
LIN {X 0,Y 369.028,Z 604.519,A -85,B 0,C 180,E1 -12793.772,E2 -12793.772} C_VEL
LIN {X 0,Y 368.992,Z 604.525,A -85,B 0,C 180,E1 -12797.768,E2 -12797.768} C_VEL
LIN {X 0,Y 368.92,Z 604.528,A -85,B 0,C 180,E1 -12801.22,E2 -12801.22} C_VEL
LIN {X 0,Y 368.948,Z 604.523,A -85,B 0,C 180,E1 -12804.775,E2 -12804.775} C_VEL
LIN {X 0,Y 368.978,Z 604.521,A -85,B 0,C 180,E1 -12808.436,E2 -12808.436} C_VEL
LIN {X 0,Y 368.901,Z 604.534,A -85,B 0,C 180,E1 -12812.237,E2 -12812.237} C_VEL
LIN {X 0,Y 368.921,Z 604.527,A -85,B 0,C 180,E1 -12815.002,E2 -12815.002} C_VEL
LIN {X 0,Y 368.906,Z 604.53,A -85,B 0,C 180,E1 -12818.641,E2 -12818.641} C_VEL
LIN {X 0,Y 368.944,Z 604.528,A -85,B 0,C 180,E1 -12822.022,E2 -12822.022} C_VEL
LIN {X 0,Y 368.918,Z 604.527,A -85,B 0,C 180,E1 -12825.183,E2 -12825.183} C_VEL
LIN {X 0,Y 368.902,Z 604.534,A -85,B 0,C 180,E1 -12828.182,E2 -12828.182} C_VEL
LIN {X 0,Y 368.904,Z 604.529,A -85,B 0,C 180,E1 -12831.36,E2 -12831.36} C_VEL
LIN {X 0,Y 368.931,Z 604.526,A -85,B 0,C 180,E1 -12835.147,E2 -12835.147} C_VEL
LIN {X 0,Y 368.923,Z 604.528,A -85,B 0,C 180,E1 -12839.047,E2 -12839.047} C_VEL
LIN {X 0,Y 368.958,Z 604.526,A -85,B 0,C 180,E1 -12842.797,E2 -12842.797} C_VEL
LIN {X 0,Y 368.94,Z 604.526,A -85,B 0,C 180,E1 -12846.113,E2 -12846.113} C_VEL
LIN {X 0,Y 368.932,Z 604.525,A -85,B 0,C 180,E1 -12849.947,E2 -12849.947} C_VEL
LIN {X 0,Y 368.972,Z 604.521,A -85,B 0,C 180,E1 -12853.399,E2 -12853.399} C_VEL
LIN {X 0,Y 369.054,Z 604.516,A -85,B 0,C 180,E1 -12856.79,E2 -12856.79} C_VEL
LIN {X 0,Y 369.064,Z 604.509,A -85,B 0,C 180,E1 -12860.132,E2 -12860.132} C_VEL
LIN {X 0,Y 369.158,Z 604.498,A -85,B 0,C 180,E1 -12862.342,E2 -12862.342} C_VEL
LIN {X 0,Y 369.139,Z 604.502,A -85,B 0,C 180,E1 -12864.538,E2 -12864.538} C_VEL
LIN {X 0,Y 369.316,Z 604.478,A -85,B 0,C 180,E1 -12867.819,E2 -12867.819} C_VEL
LIN {X 0,Y 369.456,Z 604.46,A -85,B 0,C 180,E1 -12870,E2 -12870} C_VEL
LIN {X 0,Y 369.316,Z 604.477,A -85,B 0,C 180,E1 -12872.181,E2 -12872.181} C_VEL
LIN {X 0,Y 369.195,Z 604.493,A -85,B 0,C 180,E1 -12876.558,E2 -12876.558} C_VEL
LIN {X 0,Y 369.064,Z 604.51,A -85,B 0,C 180,E1 -12879.868,E2 -12879.868} C_VEL
LIN {X 0,Y 369.033,Z 604.515,A -85,B 0,C 180,E1 -12883.772,E2 -12883.772} C_VEL
LIN {X 0,Y 368.997,Z 604.523,A -85,B 0,C 180,E1 -12887.768,E2 -12887.768} C_VEL
LIN {X 0,Y 368.99,Z 604.683,A -85,B 0,C 180,E1 -12891.875,E2 -12891.875} C_VEL
LIN {X 0,Y 370.194,Z 610.893,A -85,B 0,C 180,E1 -12893.687,E2 -12893.687} C_VEL
LIN {X 0,Y 374.232,Z 623.019,A -85,B 0,C 180,E1 -12894.172,E2 -12894.172} C_VEL
LIN {X 0,Y 376.599,Z 634.547,A -85,B 0,C 180,E1 -12894.547,E2 -12894.547} C_VEL
LIN {X 0,Y 374.953,Z 717.722,A -85,B 0,C 180,E1 -12896.254,E2 -12896.254} C_VEL
LIN {X 0,Y 374.879,Z 719.998,A -85,B 0,C 180,E1 -12896.323,E2 -12896.323} C_VEL
LIN {X 0,Y 374.236,Z 725.758,A -85,B 0,C 180,E1 -12896.496,E2 -12896.496} C_VEL
LIN {X 0,Y 371.114,Z 735.015,A -85,B 0,C 180,E1 -12896.768,E2 -12896.768} C_VEL
LIN {X 0,Y 367.713,Z 744.021,A -85,B 0,C 180,E1 -12897.153,E2 -12897.153} C_VEL
LIN {X 0,Y 366.644,Z 749.392,A -85,B 0,C 180,E1 -12897.502,E2 -12897.502} C_VEL
LIN {X 0,Y 365.838,Z 761.342,A -85,B 0,C 180,E1 -12898.512,E2 -12898.512} C_VEL
LIN {X 0,Y 364.856,Z 771.952,A -85,B 0,C 180,E1 -12899.638,E2 -12899.638} C_VEL
LIN {X 0,Y 363.977,Z 781.805,A -85,B 0,C 180,E1 -12900.936,E2 -12900.936} C_VEL
LIN {X 0,Y 363.212,Z 789.836,A -85,B 0,C 180,E1 -12902.228,E2 -12902.228} C_VEL
LIN {X 0,Y 362.33,Z 798.04,A -85,B 0,C 180,E1 -12903.841,E2 -12903.841} C_VEL
LIN {X 0,Y 361.62,Z 805.423,A -85,B 0,C 180,E1 -12905.664,E2 -12905.664} C_VEL
LIN {X 0,Y 361.149,Z 811.106,A -85,B 0,C 180,E1 -12907.453,E2 -12907.453} C_VEL
LIN {X 0,Y 360.715,Z 815.706,A -85,B 0,C 180,E1 -12909.381,E2 -12909.381} C_VEL
LIN {X 0,Y 360.43,Z 819.221,A -85,B 0,C 180,E1 -12911.525,E2 -12911.525} C_VEL
LIN {X 0,Y 360.233,Z 821.244,A -85,B 0,C 180,E1 -12913.793,E2 -12913.793} C_VEL
LIN {X 0,Y 360.202,Z 821.687,A -85,B 0,C 180,E1 -12915.381,E2 -12915.381} C_VEL
LIN {X 0,Y 360.292,Z 821.299,A -85,B 0,C 180,E1 -12916.944,E2 -12916.944} C_VEL
LIN {X 0,Y 360.435,Z 820.148,A -85,B 0,C 180,E1 -12918.475,E2 -12918.475} C_VEL
LIN {X 0,Y 360.801,Z 817.275,A -85,B 0,C 180,E1 -12920.616,E2 -12920.616} C_VEL
LIN {X 0,Y 361.152,Z 814.095,A -85,B 0,C 180,E1 -12922.196,E2 -12922.196} C_VEL
LIN {X 0,Y 361.82,Z 808.152,A -85,B 0,C 180,E1 -12924.359,E2 -12924.359} C_VEL
LIN {X 0,Y 362.561,Z 801.675,A -85,B 0,C 180,E1 -12926.149,E2 -12926.149} C_VEL
LIN {X 0,Y 363.439,Z 794.39,A -85,B 0,C 180,E1 -12927.752,E2 -12927.752} C_VEL
LIN {X 0,Y 364.55,Z 785.726,A -85,B 0,C 180,E1 -12929.278,E2 -12929.278} C_VEL
LIN {X 0,Y 365.567,Z 776.216,A -85,B 0,C 180,E1 -12930.645,E2 -12930.645} C_VEL
LIN {X 0,Y 366.623,Z 765.769,A -85,B 0,C 180,E1 -12931.858,E2 -12931.858} C_VEL
LIN {X 0,Y 367.613,Z 755.352,A -85,B 0,C 180,E1 -12932.82,E2 -12932.82} C_VEL
LIN {X 0,Y 368.504,Z 743.378,A -85,B 0,C 180,E1 -12933.682,E2 -12933.682} C_VEL
LIN {X 0,Y 369.188,Z 729.984,A -85,B 0,C 180,E1 -12934.394,E2 -12934.394} C_VEL
LIN {X 0,Y 369.707,Z 716.56,A -85,B 0,C 180,E1 -12934.847,E2 -12934.847} C_VEL
LIN {X 0,Y 371.632,Z 636.442,A -85,B 0,C 180,E1 -12936.561,E2 -12936.561} C_VEL
LIN {X 0,Y 369.604,Z 627.789,A -85,B 0,C 180,E1 -12936.91,E2 -12936.91} C_VEL
LIN {X 0,Y 363.566,Z 613.119,A -85,B 0,C 180,E1 -12937.721,E2 -12937.721} C_VEL
